//			(*Pierwsze szukanie*)
//			IF NOT bScrew1MinFound THEN															(*W1*)
//				IF ABS(ABS(lrStartPosition1FindingScrew)-ABS(Screwing1AxisRef.NcToPlc.ActPos))	>	100  THEN 
//					//IF lrScrewer1ActualTorque > (lrScrewer1MinTorqueWhenFindingScrew - 5) AND lrScrewer1ActualTorque < (lrScrewer1MaxTorqueWhenFindingScrew + 15) THEN		
////					IF diSensorHeightCV < -39000 THEN		(*W2*) //Dla Słoików 300ml
//					IF diSensorHeightCV < ((lrScrewerMaxSensorHeightWhenFindingScrew+lrScrewerMinSensorHeightWhenFindingScrew)/2) THEN		(*W2*) //Dla Słoików 300ml						
//						bScrew1MinFound						:=	TRUE;
//						lrStartPosition1FindingScrew 		:=	Screwing1AxisRef.NcToPlc.ActPos;
//					END_IF	
//				END_IF
//			END_IF
//			IF NOT bScrew2MinFound THEN															(*W1*)
//				IF ABS(ABS(lrStartPosition2FindingScrew)-ABS(Screwing2AxisRef.NcToPlc.ActPos))	>	100  THEN 
////					IF diSensorHeightCV < -39000 THEN		(*W2*)	//Dla Słoików 300ml	
//					IF diSensorHeightCV < ((lrScrewerMaxSensorHeightWhenFindingScrew+lrScrewerMinSensorHeightWhenFindingScrew)/2) THEN		(*W2*)	//Dla Słoików 300ml	
//						bScrew2MinFound						:=	TRUE;	
//						lrStartPosition2FindingScrew 		:=	Screwing2AxisRef.NcToPlc.ActPos;
//					END_IF	
//				END_IF	
//			END_IF
//			lrScrewerOffsetSensorHeightWhenFindingScrew	:=	((lrScrewerMaxSensorHeightWhenFindingScrew+lrScrewerMinSensorHeightWhenFindingScrew)/2)
//																+(lrScrewerMinSensorHeightWhenFindingScrew-lrScrewerMaxSensorHeightWhenFindingScrew)/6;
			
//			(*Drugie szukanie*)																					(*W3*)
//			IF bScrew1MinFound AND ABS(ABS(lrStartPosition1FindingScrew)-ABS(Screwing1AxisRef.NcToPlc.ActPos))	>	10  THEN 
				
//				IF diSensorHeightCV > lrScrewerOffsetSensorHeightWhenFindingScrew THEN		(*W4*)	//Dla Słoików 300ml
//					bScrew1Found						:=	TRUE;
//					mcScrewer1MoveRelative.Execute		:=	FALSE;
//					lrStartPosition1FindingScrew 		:=	Screwing1AxisRef.NcToPlc.ActPos;
//				END_IF
//			END_IF																								(*W3*)
//			IF bScrew2MinFound AND ABS(ABS(lrStartPosition2FindingScrew)-ABS(Screwing2AxisRef.NcToPlc.ActPos))	>	10  THEN 
//				IF diSensorHeightCV > ((lrScrewerMaxSensorHeightWhenFindingScrew+lrScrewerMinSensorHeightWhenFindingScrew)/2) THEN		(*W4*)	//Dla Słoików 300ml
//					bScrew2Found						:=	TRUE;
//					mcScrewer2MoveRelative.Execute		:=	FALSE;
//					lrStartPosition2FindingScrew 		:=	Screwing1AxisRef.NcToPlc.ActPos;
//				END_IF
//			END_IF

//			IF bScrew1Found  THEN

//				uiScrewing1TorqueControl		:=	6000;
//				mcScrewer1Stop.Execute			:=	TRUE;
				
//			END_IF
			
//			IF bScrew2Found  THEN

//				uiScrewing2TorqueControl		:=	6000;
//				mcScrewer2Stop.Execute			:=	TRUE;
//			END_IF			
			
//			IF	((bScrew1Found AND mcScrewer1Stop.Done) OR NOT bRun1 OR mcScrewer1MoveRelative.Done) AND
//				((bScrew2Found AND mcScrewer2Stop.Done) OR NOT bRun2 OR mcScrewer2MoveRelative.Done)
//			THEN
//				 mcScrewer1MoveRelative.Execute 	:=	FALSE;
//				 mcScrewer1Stop.Execute				:=	FALSE;
//				 mcScrewer2MoveRelative.Execute 	:=	FALSE;		
//				 mcScrewer2Stop.Execute				:=	FALSE;	 
//				 iFindingScrewCASE					:=	iFindingScrewCASE	+	10;	
//			END_IF
			
//		50: 
//			IF tonFindingScrewDelay.Q THEN
// 				iFindingScrewCASE					:=	iFindingScrewCASE	+	10;						
//			END_IF




END_IF
END_ACTION

ACTION Running6ScrewingMomentaryMode:
IF mcScrewer1TorqueControl.Error OR mcScrewer1MoveVelocity.Error OR mcScrewer1MoveVelocity2.Error
	 OR mcScrewer1MoveVelocity3.Error OR mcScrewer1MoveRelative.Error OR mcScrewer1MoveAbsolute.Error THEN
	bTest:= TRUE;
END_IF
tonInEndVelocity(IN:=mcScrewer1MoveContinuousRel.InEndVelocity, PT:=T#2MS);


				(********** TRYB MOMENTOWY **********)
					CASE iScrewingCase OF 	
					0:
						(* Wersja 2 - gearowanie Multi Master***************************************************************) 
						IF iTool <> 2 THEN
							bGripper1Actuator						:=	bRun1; // Ponowne załączanie chwytaków, dlatego
							bGripper2Actuator						:=	bRun2; // że jest możliwa duża ilość opcji
						ELSE
							bGripper1Actuator						:=	FALSE; // Ponowne załączanie chwytaków, dlatego
							bGripper2Actuator						:=	FALSE;
						END_IF
						//Właczenie sięcia osi
						mcHeightGearInMultiMaster.Enable			:=	TRUE;				
						//Jak osie spięte to początek kręcenia
						IF	mcHeightGearInMultiMaster.InGear AND 
							(tonGripper1Delay.Q OR sTool = 'ksztaltowa/do kulek' OR NOT bRun1) AND (tonGripper2Delay.Q OR sTool = 'ksztaltowa/do kulek'  OR NOT bRun2) // ton'y powinny być już wczesniej załączone jeżeli były chwytaki	
						THEN
							//Bloczek obrotu o zadany kąt i kontynuowania ruchu z zadaną prędkością
							mcScrewer1MoveContinuousRel.Execute				:= bRun1;
							//Kąt zmodyfikowany o różnicę między pozycją zatrzymania zakręcarki a pozycją wykrycia gwintu
							mcScrewer1MoveContinuousRel.Distance			:= Screwing1AxisRef.NcToPlc.ActPos - lrStartPosition1 + lrPackageTurnoversToFullScrewed*360.0-30.0;

							//DODAĆ ZABEZPIECZENIE JAK WYJDZIE ABSURDALNY KĄT
							
							//Prędkość na wyjściu z bloczka 120RPM - Inercja zakręcarki jest rozsądna
							mcScrewer1MoveContinuousRel.EndVelocity			:= 360*2;
							//Prędkość zakręcania wg parametrów
							mcScrewer1MoveContinuousRel.Velocity			:= (lrScrewerSpeed);
														
							iScrewingCase									:=	25;//iScrewingCase + 10;			
						END_IF
						
					10:	
					
						IF ABS(ABS(lrStartPosition1)-ABS(Screwing1AxisRef.NcToPlc.ActPos))>(lrPackageTurnoversToFullScrewed*360.0-90.0)  THEN 
							mcScrewer1MoveVelocity.Execute					:= FALSE;
							mcScrewer1MoveVelocity2.Execute					:= bRun1;
							mcScrewer1MoveVelocity2.Velocity				:= 360;
							uiScrewing1TorqueControl						:=	60000;
						//	mcScrewer1TorqueControl.Torque					:=	-5000;		
						//	mcScrewer1TorqueControl.TorqueRamp				:=	80000;	
							mcScrewer1TorqueControl.VelocityLimitHigh		:=	360;//(lrScrewerSpeed)/3.0;
							mcScrewer1TorqueControl.VelocityLimitLow		:=	-360;//-(lrScrewerSpeed)/3.0;
							iScrewingCase									:=	iScrewingCase + 10;	
						END_IF	
							
//						IF ABS(ABS(lrStartPosition2)-ABS(Screwing2AxisRef.NcToPlc.ActPos))>(lrPackageTurnoversToFullScrewed*360.0/7)  THEN 
//							mcScrewer2TorqueControl.Torque					:=	-9;		
//							mcScrewer2TorqueControl.TorqueRamp				:=	1500;					
//							mcScrewer2TorqueControl.VelocityLimitLow		:=	-4000;
//						END_IF	
					20:	
						mcScrewer1MoveVelocity2.Execute					:= FALSE;
						IF ABS(ABS(lrStartPosition1)-ABS(Screwing1AxisRef.NcToPlc.ActPos))>(lrPackageTurnoversToFullScrewed*360.0-15.0)  THEN
							mcScrewer1MoveVelocity2.Execute					:= FALSE;
							mcScrewer1TorqueControl.Execute					:=	bRun1;
							mcScrewer1TorqueControl.Torque					:=	(INT_TO_UINT(iScrewer1SetTorque)+iScrewer1AddTorque);		
						//	mcScrewer1TorqueControl.TorqueRamp				:=	4000;					
						//	mcScrewer1TorqueControl.VelocityLimitLow		:=	- 10;//(lrScrewerSpeed)/3.0;
							iScrewingCase									:=	iScrewingCase + 10;	
						END_IF	
							
						IF ABS(ABS(lrStartPosition2)-ABS(Screwing2AxisRef.NcToPlc.ActPos))>(lrPackageTurnoversToFullScrewed*360.0/6)  THEN 
							mcScrewer2TorqueControl.Torque					:=	(INT_TO_UINT(iScrewer2SetTorque)+iScrewer2AddTorque);		
							mcScrewer2TorqueControl.TorqueRamp				:=	4000;					
							mcScrewer2TorqueControl.VelocityLimitLow		:=	-(lrScrewerSpeed);
						END_IF	
						
					25:
						//Jak dojedzie do końca ruchu
						IF mcScrewer1MoveContinuousRel.InEndVelocity AND tonInEndVelocity.Q THEN
							mcScrewer1MoveContinuousRel.Execute				:= FALSE;
							//Przygotowanie trybu momentowego
							mcScrewer1TorqueControl.Execute					:=	bRun1;
							mcScrewer1TorqueControl.Torque					:=	(INT_TO_UINT(iScrewer1SetTorque)+iScrewer1AddTorque);	
							mcScrewer1TorqueControl.TorqueRamp				:=	8000;
							mcScrewer1TorqueControl.VelocityLimitHigh		:=	360*2;//(lrScrewerSpeed)/3.0;
							mcScrewer1TorqueControl.VelocityLimitLow		:=	-360*2;//-(lrScrewerSpeed)/3.0;	
							iScrewingCase									:=	30;//iScrewingCase + 10;	
						END_IF
	
					30:
						IF tonMomentaryScrewing1Timer.Q OR bWarning1 THEN
							mcScrewer1Stop.Execute				:=	TRUE;
							bGripper1Actuator					:=	FALSE;
							mcScrewer1TorqueControl.Execute		:=	FALSE;
							uiScrewing1TorqueControl			:=	0;
							bScrewed1							:=	TRUE;	
						END_IF
						IF tonMomentaryScrewing2Timer.Q OR bWarning2 THEN
							mcScrewer2Stop.Execute				:=	TRUE;
							bGripper2Actuator					:=	FALSE;
							mcScrewer2TorqueControl.Execute		:=	FALSE;
							uiScrewing2TorqueControl			:=	0;
							bScrewed2							:=	TRUE;		
						END_IF
				
						// Warunki zakręcenia zaleznie od uruchomionej zakręcarki
						IF (bScrewed1 OR NOT bRun1) AND (bScrewed2 OR NOT bRun2) AND
							(mcScrewer1Stop.Done OR NOT mcScrewer1Stop.Execute) AND 
							(mcScrewer2Stop.Done OR NOT mcScrewer2Stop.Execute) THEN
								mcScrewer1Stop.Execute			:= FALSE;
								mcScrewer2Stop.Execute			:= FALSE;
								iScrewingCase					:= iScrewingCase + 10;		
						END_IF
					40:
						(* Rozgearowanie osi *)
						mcHeightGearOut.Execute				:=	TRUE;
						mcHeightGearInMultiMaster.Enable	:=	FALSE;
	
						IF  mcHeightGearOut.Done THEN
							mcHeightGearOut.Execute					:= FALSE;
							eRunningState							:= E_GripperScrewer.eHolding;	
							iScrewingCase							:= 0;	
						END_IF			
					END_CASE
END_ACTION

ACTION Running6ScrewingPositionTorqueMode:
				(********* TRYB POZYCYJNY  *********)
				
				lrPackageThreadPitch;	
				(*Wymuszanie zwiększonego momentu przez 1/4 całego zakręcania*)
				IF ABS(ABS(lrStartPosition1)-ABS(Screwing1AxisRef.NcToPlc.ActPos))>(lrPackageTurnoversToFullScrewed*360.0/7)  THEN 
							uiScrewing1TorqueControl			:=	(INT_TO_UINT(iScrewer1SetTorque+3)*10)+(iScrewer1AddTorque*10);	
				ELSE		uiScrewing1TorqueControl			:=	6000;
				END_IF
				//uiScrewing1TorqueControl			:=	(INT_TO_UINT(iScrewerSetTorque+3)*10)+iScrewer1AddTorque;	
				(*Wymuszanie zwiększonego momentu przez 1/4 całego zakręcania*)
				IF ABS(ABS(lrStartPosition2)-ABS(Screwing2AxisRef.NcToPlc.ActPos))>(lrPackageTurnoversToFullScrewed*360.0/7)  THEN 
							uiScrewing2TorqueControl			:=	(INT_TO_UINT(iScrewer2SetTorque+3)*10)+(iScrewer2AddTorque*10);		
				ELSE		uiScrewing2TorqueControl			:=	6000;
				END_IF	

					CASE iScrewingCase OF 	
					0:
						(* Wersja 2 - gearowanie Multi Master***************************************************************) 
						IF iTool <> 2 THEN
							bGripper1Actuator						:=	bRun1; // Ponowne załączanie chwytaków, dlatego
							bGripper2Actuator						:=	bRun2; // że jest możliwa duża ilość opcji
						ELSE
							bGripper1Actuator						:=	FALSE; // Ponowne załączanie chwytaków, dlatego
							bGripper2Actuator						:=	FALSE; // że jest możliwa duża ilość opcji
						END_IF
						mcHeightGearInMultiMaster.Enable			:=	TRUE;				
						(* Start zakręcania *)
						IF	mcHeightGearInMultiMaster.InGear AND 
							(tonGripper1Delay.Q OR sTool = 'ksztaltowa/do kulek' OR NOT bRun1) AND (tonGripper2Delay.Q OR sTool = 'ksztaltowa/do kulek' OR NOT bRun2) // ton'y powinny być już wczesniej załączone jeżeli były chwytaki	
						THEN

							CASE iScrewing2Case OF 	
								
							0:
							
								mcScrewer1MoveVelocity2.Velocity		:=	5000;
								mcScrewer1MoveVelocity2.Execute		:=	bRun1;
								mcScrewer1MoveVelocity2.Direction	:=	MC_Positive_Direction;
																				
								mcScrewer2MoveVelocity2.Velocity		:=	5000;
								mcScrewer2MoveVelocity2.Execute		:=	bRun2;
								mcScrewer2MoveVelocity2.Direction	:=	MC_Positive_Direction;	
	
								iScrewing2Case						:=	iScrewing2Case + 10;										
							
							10:
								mcScrewer1MoveVelocity2.Execute		:=	FALSE;
								mcScrewer2MoveVelocity2.Execute		:=	FALSE;
							
								iScrewing2Case						:=	iScrewing2Case + 10;
	
							20:
							
								mcScrewer1MoveVelocity.Velocity		:=	lrScrewerSpeed;		
								mcScrewer1MoveVelocity.Direction	:=	MC_Positive_Direction;	
								IF ABS(ABS(lrStartPosition1)-ABS(Screwing1AxisRef.NcToPlc.ActPos))>(lrPackageTurnoversToFullScrewed*360.0/7)  THEN 									
									mcScrewer1MoveVelocity.Execute		:=	bRun1;									
								END_IF
								mcScrewer2MoveVelocity.Velocity		:=	lrScrewerSpeed;	
								mcScrewer1MoveVelocity.Direction		:=	MC_Positive_Direction;	
								IF ABS(ABS(lrStartPosition2)-ABS(Screwing2AxisRef.NcToPlc.ActPos))>(lrPackageTurnoversToFullScrewed*360.0/7)  THEN 
	
									mcScrewer2MoveVelocity.Execute		:=	bRun2;
								END_IF			

								IF (mcScrewer1MoveVelocity.Execute OR NOT bRun1) AND (mcScrewer2MoveVelocity.Execute OR NOT bRun2) THEN
									iScrewing2Case					:= 0	;
									iScrewingCase					:= iScrewingCase + 10;		
								END_IF
								
							END_CASE
							
						END_IF
						
					10:	
					
						(*Zmniejszanie prędkości jeżeli jest już przytrzymanie*)
						IF tonTightScrewing1Timer.ET > T#0S AND Screwing1AxisRef.NcToPlc.ActVelo < 10 THEN
							//mcScrewer1MoveVelocity.Execute		:= FALSE;
							//mcScrewer1MoveVelocity2.Execute		:= FALSE;
							
							//mcScrewer1MoveVelocity3.Velocity	:=	10;
							//mcScrewer1MoveVelocity3.Execute		:=	bRun1;
							//mcScrewer1MoveVelocity3.Direction	:=	MC_Positive_Direction;		

							rScrewing1ProportionalGain	:= 0;
							//rScrewing2ProportionalGain	:= 0;												
						END_IF
						
						IF tonTightScrewing2Timer.ET > T#0S AND Screwing2AxisRef.NcToPlc.ActVelo < 10 THEN
							//mcScrewer2MoveVelocity.Execute		:= FALSE;
							//mcScrewer2MoveVelocity2.Execute		:= FALSE;
							
							//mcScrewer2MoveVelocity3.Velocity	:=	10;
							//mcScrewer2MoveVelocity3.Execute		:=	bRun1;
							//mcScrewer2MoveVelocity3.Direction	:=	MC_Positive_Direction;		

							//rScrewing1ProportionalGain	:= 0;
							rScrewing2ProportionalGain	:= 0;												
						END_IF					
					
						(* Sprawdzanie czy osiągnięto moment lub zbyt długie zakracanie*)				
						IF tonTightScrewing1Timer.Q OR bWarning1 THEN
							bGripper1Actuator					:=	FALSE;
							bScrewed1							:=	TRUE;	
						END_IF
						IF tonTightScrewing2Timer.Q OR bWarning2 THEN
							bGripper2Actuator					:=	FALSE;
							bScrewed2							:=	TRUE;		
						END_IF
	
						IF tonTightScrewing1TimerAndOpenedGripper.Q THEN
							mcScrewer1Stop.Execute				:=	TRUE;
							mcScrewer1MoveVelocity.Execute		:=	FALSE;
							mcScrewer1MoveVelocity2.Execute		:=	FALSE;
							mcScrewer1MoveVelocity3.Execute		:=	FALSE;							
							uiScrewing1TorqueControl			:=	0;
						END_IF
						IF tonTightScrewing2TimerAndOpenedGripper.Q THEN
							mcScrewer2Stop.Execute				:=	TRUE;
							mcScrewer2MoveVelocity.Execute		:=	FALSE;
							mcScrewer2MoveVelocity2.Execute		:=	FALSE;	
							mcScrewer2MoveVelocity3.Execute		:=	FALSE;							
							uiScrewing2TorqueControl			:=	0;
						END_IF
					
						// Warunki zakręcenia zaleznie od uruchomionej zakręcarki
						IF (tonTightScrewing1TimerAndOpenedGripper.Q OR NOT bRun1) AND (tonTightScrewing2TimerAndOpenedGripper.Q OR NOT bRun2) AND
							(mcScrewer1Stop.Done OR NOT mcScrewer1Stop.Execute) AND 
							(mcScrewer2Stop.Done OR NOT mcScrewer2Stop.Execute) THEN
								mcScrewer1Stop.Execute			:= FALSE;
								mcScrewer2Stop.Execute			:= FALSE;
								iScrewingCase					:= iScrewingCase + 10;		
						END_IF
						
					20:
						(* Rozgearowanie osi *)
						mcHeightGearOut.Execute				:=	TRUE;
						mcHeightGearInMultiMaster.Enable	:=	FALSE;
	
						IF  mcHeightGearOut.Done THEN
							mcHeightGearOut.Execute					:= FALSE;
							eRunningState							:= E_GripperScrewer.eHolding;	
							iScrewingCase							:= 0;	
						END_IF			
					END_CASE
END_ACTION

ACTION Screwer1ControlBlocks:
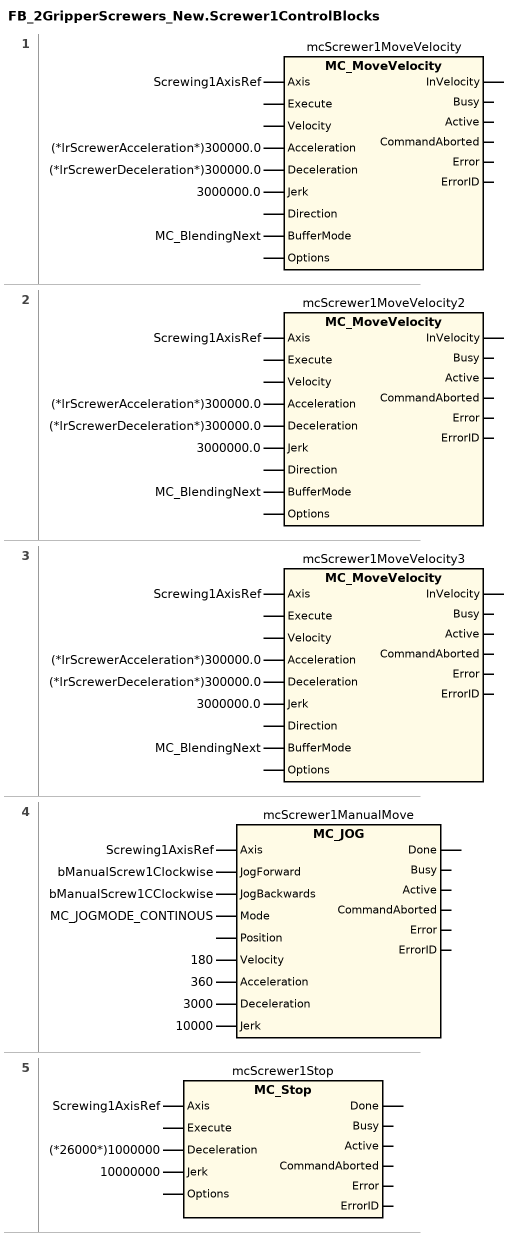
// NETWORK 1
mcScrewer1MoveVelocity(
    Axis := Screwing1AxisRef,
    Acceleration := (*lrScrewerAcceleration*)300000.0,
    Deceleration := (*lrScrewerDeceleration*)300000.0,
    Jerk := 3000000.0,
    BufferMode := MC_BlendingNext); // MC_MoveVelocity

// NETWORK 2
mcScrewer1MoveVelocity2(
    Axis := Screwing1AxisRef,
    Acceleration := (*lrScrewerAcceleration*)300000.0,
    Deceleration := (*lrScrewerDeceleration*)300000.0,
    Jerk := 3000000.0,
    BufferMode := MC_BlendingNext); // MC_MoveVelocity

// NETWORK 3
mcScrewer1MoveVelocity3(
    Axis := Screwing1AxisRef,
    Acceleration := (*lrScrewerAcceleration*)300000.0,
    Deceleration := (*lrScrewerDeceleration*)300000.0,
    Jerk := 3000000.0,
    BufferMode := MC_BlendingNext); // MC_MoveVelocity

// NETWORK 4
mcScrewer1ManualMove(
    Axis := Screwing1AxisRef,
    JogForward := bManualScrew1Clockwise,
    JogBackwards := bManualScrew1CClockwise,
    Mode := MC_JOGMODE_CONTINOUS,
    Velocity := 180,
    Acceleration := 360,
    Deceleration := 3000,
    Jerk := 10000); // MC_JOG

// NETWORK 5
mcScrewer1Stop(Axis := Screwing1AxisRef, Deceleration := (*26000*)1000000, Jerk := 10000000); // MC_Stop

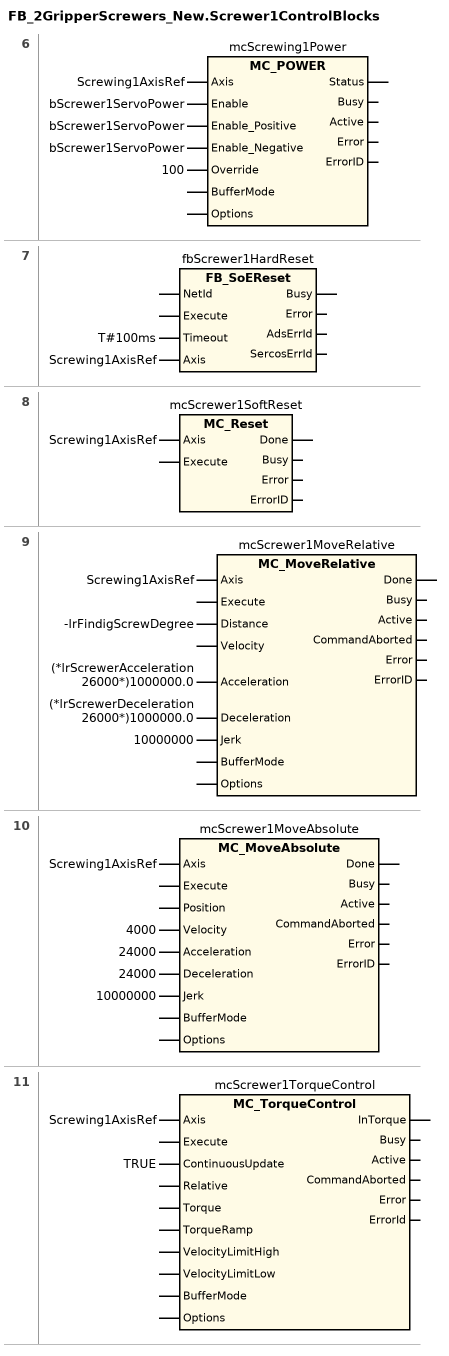
// NETWORK 6
mcScrewing1Power(
    Axis := Screwing1AxisRef,
    Enable := bScrewer1ServoPower,
    Enable_Positive := bScrewer1ServoPower,
    Enable_Negative := bScrewer1ServoPower,
    Override := 100); // MC_POWER

// NETWORK 7
fbScrewer1HardReset(Timeout := T#100ms, Axis := Screwing1AxisRef); // FB_SoEReset

// NETWORK 8
mcScrewer1SoftReset(Axis := Screwing1AxisRef); // MC_Reset

// NETWORK 9
mcScrewer1MoveRelative(
    Axis := Screwing1AxisRef,
    Distance := -lrFindigScrewDegree,
    Acceleration := (*lrScrewerAcceleration 26000*)1000000.0,
    Deceleration := (*lrScrewerDeceleration 26000*)1000000.0,
    Jerk := 10000000); // MC_MoveRelative

// NETWORK 10
mcScrewer1MoveAbsolute(
    Axis := Screwing1AxisRef,
    Velocity := 4000,
    Acceleration := 24000,
    Deceleration := 24000,
    Jerk := 10000000); // MC_MoveAbsolute

// NETWORK 11
mcScrewer1TorqueControl(Axis := Screwing1AxisRef, ContinuousUpdate := TRUE); // MC_TorqueControl

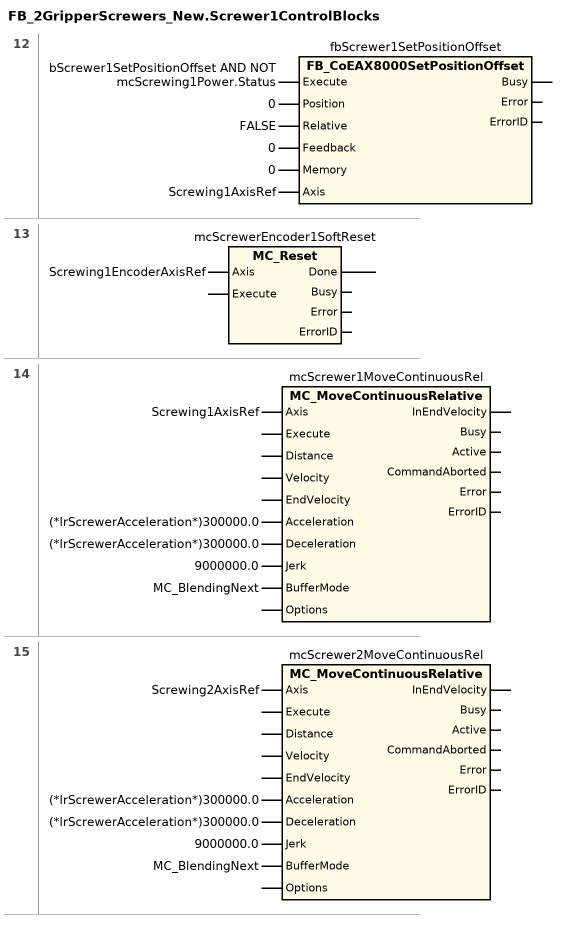
// NETWORK 12
fbScrewer1SetPositionOffset(
    Execute := bScrewer1SetPositionOffset AND NOT mcScrewing1Power.Status,
    Position := 0,
    Relative := FALSE,
    Feedback := 0,
    Memory := 0,
    Axis := Screwing1AxisRef); // FB_CoEAX8000SetPositionOffset

// NETWORK 13
mcScrewerEncoder1SoftReset(Axis := Screwing1EncoderAxisRef); // MC_Reset

// NETWORK 14
mcScrewer1MoveContinuousRel(
    Axis := Screwing1AxisRef,
    Acceleration := (*lrScrewerAcceleration*)300000.0,
    Deceleration := (*lrScrewerAcceleration*)300000.0,
    Jerk := 9000000.0,
    BufferMode := MC_BlendingNext); // MC_MoveContinuousRelative

// NETWORK 15
mcScrewer2MoveContinuousRel(
    Axis := Screwing2AxisRef,
    Acceleration := (*lrScrewerAcceleration*)300000.0,
    Deceleration := (*lrScrewerAcceleration*)300000.0,
    Jerk := 9000000.0,
    BufferMode := MC_BlendingNext); // MC_MoveContinuousRelative
END_ACTION

ACTION Screwer2ControlBlocks:
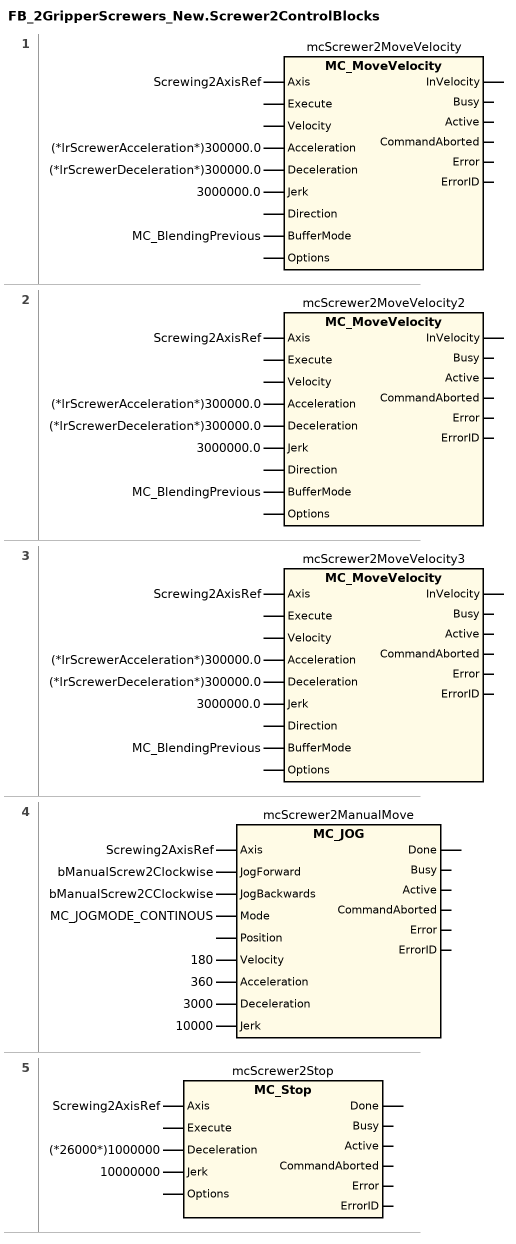
// NETWORK 1
mcScrewer2MoveVelocity(
    Axis := Screwing2AxisRef,
    Acceleration := (*lrScrewerAcceleration*)300000.0,
    Deceleration := (*lrScrewerDeceleration*)300000.0,
    Jerk := 3000000.0,
    BufferMode := MC_BlendingPrevious); // MC_MoveVelocity

// NETWORK 2
mcScrewer2MoveVelocity2(
    Axis := Screwing2AxisRef,
    Acceleration := (*lrScrewerAcceleration*)300000.0,
    Deceleration := (*lrScrewerDeceleration*)300000.0,
    Jerk := 3000000.0,
    BufferMode := MC_BlendingPrevious); // MC_MoveVelocity

// NETWORK 3
mcScrewer2MoveVelocity3(
    Axis := Screwing2AxisRef,
    Acceleration := (*lrScrewerAcceleration*)300000.0,
    Deceleration := (*lrScrewerDeceleration*)300000.0,
    Jerk := 3000000.0,
    BufferMode := MC_BlendingPrevious); // MC_MoveVelocity

// NETWORK 4
mcScrewer2ManualMove(
    Axis := Screwing2AxisRef,
    JogForward := bManualScrew2Clockwise,
    JogBackwards := bManualScrew2CClockwise,
    Mode := MC_JOGMODE_CONTINOUS,
    Velocity := 180,
    Acceleration := 360,
    Deceleration := 3000,
    Jerk := 10000); // MC_JOG

// NETWORK 5
mcScrewer2Stop(Axis := Screwing2AxisRef, Deceleration := (*26000*)1000000, Jerk := 10000000); // MC_Stop

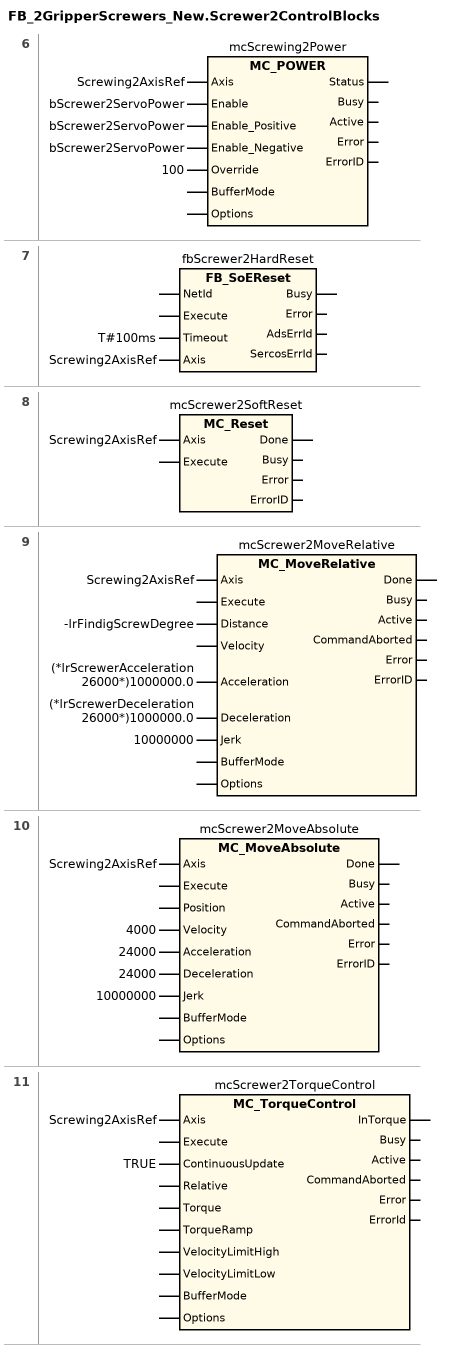
// NETWORK 6
mcScrewing2Power(
    Axis := Screwing2AxisRef,
    Enable := bScrewer2ServoPower,
    Enable_Positive := bScrewer2ServoPower,
    Enable_Negative := bScrewer2ServoPower,
    Override := 100); // MC_POWER

// NETWORK 7
fbScrewer2HardReset(Timeout := T#100ms, Axis := Screwing2AxisRef); // FB_SoEReset

// NETWORK 8
mcScrewer2SoftReset(Axis := Screwing2AxisRef); // MC_Reset

// NETWORK 9
mcScrewer2MoveRelative(
    Axis := Screwing2AxisRef,
    Distance := -lrFindigScrewDegree,
    Acceleration := (*lrScrewerAcceleration 26000*)1000000.0,
    Deceleration := (*lrScrewerDeceleration 26000*)1000000.0,
    Jerk := 10000000); // MC_MoveRelative

// NETWORK 10
mcScrewer2MoveAbsolute(
    Axis := Screwing2AxisRef,
    Velocity := 4000,
    Acceleration := 24000,
    Deceleration := 24000,
    Jerk := 10000000); // MC_MoveAbsolute

// NETWORK 11
mcScrewer2TorqueControl(Axis := Screwing2AxisRef, ContinuousUpdate := TRUE); // MC_TorqueControl

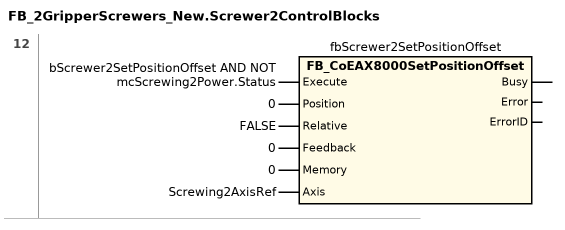
// NETWORK 12
fbScrewer2SetPositionOffset(
    Execute := bScrewer2SetPositionOffset AND NOT mcScrewing2Power.Status,
    Position := 0,
    Relative := FALSE,
    Feedback := 0,
    Memory := 0,
    Axis := Screwing2AxisRef); // FB_CoEAX8000SetPositionOffset
END_ACTION

ACTION Simulation:
(* Przyśpieszanie bloku gdy jest włączona symulacja*)

//tonSimulationScrewing1			(IN:=eRunningState=E_GripperScrewer.eScrewing 	AND bRun1 AND NOT bScrewed1 AND bSimulation,	PT:=T#0MS);
//tonSimulationScrewing2			(IN:=eRunningState=E_GripperScrewer.eScrewing 	AND bRun1 AND NOT bScrewed2 AND bSimulation,	PT:=T#0MS);

IF bSimulation THEN 			// Włączona symulacja
	tTooLongScrewing1 := T#250MS;
	tTooLongScrewing2 := T#250MS;	
ELSE							// Normalna praca
	tTooLongScrewing1 := T#2S; 	//Zmienić na 2
	tTooLongScrewing2 := T#2S;	//Zmienić na 2
END_IF
END_ACTION

ACTION Statistics:

IF LREAL_TO_INT(lrHeightEndScrewingPosition)<> LREAL_TO_INT(lrHeightReadyPosition) THEN
	rtrigCycleTimerRead(CLK:=LREAL_TO_INT(lrHeightActualPosition) = LREAL_TO_INT(lrHeightReadyPosition));
	IF rtrigCycleTimerRead.Q THEN
			tCycleTime:=tonCycleTimer.ET;
	END_IF
	tonCycleTimer(IN:=LREAL_TO_INT(lrHeightActualPosition) <> LREAL_TO_INT(lrHeightReadyPosition),PT:=T#1D);	
ELSE
	rtrigCycleTimerRead(CLK:=(eRunningState=E_GripperScrewer.eDone) OR (eRunningState=E_GripperScrewer.eNotDone));
	IF rtrigCycleTimerRead.Q THEN
		tCycleTime:=tonCycleTimer.ET;
	END_IF
	tonCycleTimer(IN:=eRunningState>E_GripperScrewer.eReady,PT:=T#1D);
END_IF
END_ACTION

ACTION Tools:
(*Narzędzia*)
AsToolDescription[0] := 'Głowica dwuszczękowa';
AsToolDescription[1] := 'Głowica trójszczękowa'; 
AsToolDescription[2] := 'Głowica kształtowa/do kulek';
AsToolDescription[3] := 'Głowica wbijająca'; 
AsToolDescription[4] := 'Głowica zasysająca';


(*Głowica wbijająca*)
IF iTool = 3 THEN
	bOptionCapPushingWithoutScrewing := TRUE;
ELSE
	bOptionCapPushingWithoutScrewing := FALSE;
END_IF

(*Przepisanie wybranego narzędzia do zmiennej typu string*)
(*!!!!! NIE ZMIENIAĆ OPISÓW, POWIĄZANE W PROGRAMIE !!!!!!*)
IF iTool = 0 THEN sTool := 'dwuszczekowa';			END_IF 
IF iTool = 1 THEN sTool := 'trojszczekowa';			END_IF
IF iTool = 2 THEN sTool := 'ksztaltowa/do kulek';	END_IF
IF iTool = 3 THEN sTool := 'wbijajaca';				END_IF
IF iTool = 4 THEN sTool := 'zasysajaca';			END_IF
END_ACTION

ACTION TorqueControl:

(*Konfiguracja MC_TorqueControl*)
//T_TorqueControlOptions;
mcScrewer1TorqueControl.Options.EnableManualTorqueStartValue := FALSE;//TRUE;
mcScrewer1TorqueControl.Options.ManualTorqueStartValue       := Screwing1AxisRef.NcToPlc.ActTorque;

mcScrewer2TorqueControl.Options.EnableManualTorqueStartValue := TRUE;
mcScrewer2TorqueControl.Options.ManualTorqueStartValue       :=  Screwing2AxisRef.NcToPlc.ActTorque;
END_ACTION

ACTION Warnings:
//Resetowanie warningów przy nastepnym cyklu

IF rtRun1.Q  OR rtRun2.Q THEN
	
	bWarning1			:=	FALSE;
	bWarning1A			:=	FALSE;
	bWarning1B			:=	FALSE;
	bWarning1C			:=	FALSE;
	bWarning1D			:=	FALSE;
	bWarning1E			:=	FALSE;	
	bWarning2			:=	FALSE;
	bWarning2A			:=	FALSE;
	bWarning2B			:=	FALSE;
	bWarning2C			:=	FALSE;
	bWarning2D			:=	FALSE;
	bWarning2E			:=	FALSE;
	udiWarningID		:=	0;
	sWarningDescription	:=	'';
END_IF
END_ACTION

END_FUNCTION_BLOCK

// ---- POUs/FB/FB_CatchStation.TcPOU
(*
Nazwa:			FB_CatchStation
Opis:			Chwytak pod stacjami 
Wersja:			v1.2
Data:			2025-07-08
Autor:			TW,DP
Urzadzenia:		Silownik chwytania, podnośnik JIESANG
Konfiguracja:	
Zmiany:
20250708 - Homing false po wyj. z Manual
20230222 - Zwieksozmny czas bledu 9

Info:
- dodano błędy od nastaw powyżej max i min (error 7 i 8)
- dodawno bHomingNeeded
- wylaczanie wyjść zmiana 2 wylaczanie wyjsc jak zniknie Enable
*)


FUNCTION_BLOCK FB_CatchStation
VAR_INPUT
	bEnable: BOOL;						//Zezwolenie na pracę
	bEStop:BOOL;						//Stop Awaryjny włączony
	bRun:BOOL;							//Rozkaz łapania 
	bHoming:BOOL;						//Zezwolenie na wykonanie bazowania i pozycjonowania podajnika
	bHeightSet:BOOL;					//Ustaw wysokość
	bChangeover:BOOL;					//Ustawianie na zadaną wysokość do wymiany elementów formatowych
	bChangeOver2:BOOL;
	bIgnoreError:BOOL;					//Ignorowania błędów cyklu pracy
	bReset:BOOL;						//Reset błędu, jeśli w stanie "eError"
	nGripperScrewerPosition   	:LREAL; // Aktualna pozycja serwa od podnoszenia
	nSafetyScrewerPosition		:LREAL;	// zadana bezpieczna pozycja 
	bScrewerbError				:BOOL;  // Sygnał błędu od zakręcarki
	nPositionHeightSV:LREAL;			//Wysokość zadana na której ma znajdować się stacja
	bOpenedActuatorSensor:BOOL;			//Czujnik otwarcia siłownika łapania
	bClosedActuatorSensor:BOOL;			//Czujnik otwarcia siłownika łapania
	lrMaxHeight:LREAL;					//Maksymalna wysokość podnośnika chwytaka
	lrMinHeight:LREAL;					//Minimalna wysokość podnośnika chwytaka
	bManualMovement:BOOL;				//Zezwolenie na ruchy ręcznę
	bUnlockColision:BOOL:=FALSE;		//Odblokowywanie możliwośći kolizji
	bAlarmSVCVDiffHeightDisable:BOOL;	//Wyłączenie alarmu od rożnicy wysokości zadanej od aktualnej
	bNoLifter:BOOL;						//Podnośnik
	
	_HEIGHTMOTOR_ :BOOL;	
				
	rHeightMotorPositionOffset :REAL;		//Wysokość bazowani podnośnika
	udiHeightMotorEncoderCV		: UDINT;
	bHeightEncoderSetCDone		: BOOL;	

	_ALARMINFO_ :BOOL;
	iStationIndex:UDINT;					//Numer stacji 
	sStationName:WSTRING;					//Nazwa stacji	

	
END_VAR
VAR_OUTPUT
	eState: E_Station;						//Stan ogólny bloku
	eRunningState: E_CatchStationState;		//Stan wewnętrzny
	bError: BOOL;							//Błąd stacji
	nErrorNr: UDINT;						//Nr błędu podajnika platynek
	sErrorDescription:STRING(200);				//Opis błędu
	sErrorDescription2: STRING(200);				//Opis błędu 2
	sErrorStationName:STRING;				//Nazwa stacji
	udiStationID: UDINT;				// Nr stacji

	bCatchActuator:BOOL;					//Sterownie siłownika łapania opakowania
	bHeightMotorUp:BOOL;					//Sterowanie silnikiem podnośnika  - RUCH W GÓRĘ
	bHeightMotorDown:BOOL;					//Sterowanie silnikiem podnośnika  - RUCH W DÓŁ
	lrHeightMotorCV:LREAL;					//Aktualna pozycja podnośnika
	tCycleTime:TIME;
	bHomingDone:BOOL;						//Wymagane ponowne bazowanie (blad podczas bazowania lub stop awaryjny)
	bCycleDone:BOOL;
	bCycleNotDone:BOOL;
	
				
	udiHeightMotorEncoderSetCV	: UDINT;	
	bHeightEncoderSetC			: BOOL;		

END_VAR
VAR
	tonHeightNoChange: TON; 			//Timer wykrycia braku ruchu siłownika zmiany wysokości stacji
	nLastPositionHeightCV: LREAL;		//Pozycja podnośnika w poprzednim cyklu programu
	tonErrorHeightChange: TON; 			//Timer błędu podnośnika
	// Czas zadziałania siłownika
	tonCatchingTime: TON;
	// Timer blokady otwierania chwytaka
	tonOpeningBlocked: TON;
	rtEncoderHomed:R_TRIG;
	tonCycleTimer:TON;
	rtrigCycleTimerRead:R_TRIG;
	
	tofMotorUpPermition: TOF;
	tofMotorDownPermition: TOF;
	tonLimitPosMinReachedDelay: TON;
	tonLimitPosMaxReachedDelay: TON;
	tonMaxHeight		: TON;
	tonMinHeight		: TON;
	tonSVCVDiffHeight	: TON;
	
	//Podnośnik Jiesang	
	fbHeightMotorEncoder: FB_JiesangActuatorEncoderModul;	// Blok enkodera podnośnika chwytaka stabilizującego pod zakręcarką	
	bHeightMotorEncoderCounterReset:BOOL; 				//Sygnał resetu enkodera
	bHeightMotorEncoderHomed:BOOL;						//Informacja od enkodera że jest zbazowany

	eLastState: E_Station;							//Stan ogólny bloku
	eLastRunningState: E_CatchStationState;			//Stan podbloku
	eLastStateTemp: E_Station;						//Stan ogólny bloku
	eLastRunningStateTemp: E_CatchStationState;		//Stan podbloku
	bStateError: BOOL;

	tonStopping: TON;
	tofHeightMotorDown: TOF;
	iCaseChangeover: INT;
	tonChangeOverLimitPosMinReachedDelay: TON;
	tonChangeoverLimitPosMaxReachedDelay: TON;
	
	//Zmienne od EVENTLOGGER
	bAlarmInit 						: BOOL := TRUE; 
	nAlarmNumerator					: INT;
	arfbAlarm						: ARRAY[0..19] OF  FB_TcAlarm;		//Tablica bloczków błędów
	fbSourceInfo 					: FB_TcSourceInfo;
	iSourceInfo						: I_TcSourceInfo;
	sAlarmTest						: STRING;
	//Koniec zmiennych od EVENTLOGGER
END_VAR

VAR_IN_OUT
	bManualCatchActuator:BOOL;		//Ruch ręczny siłownikiem podajnika platynek
	bManualHeightMotorUp:BOOL;			//Ruch ręczny podnośnika stacji w górę
	bManualHeightMotorDown:BOOL;		//Ruch ręczny podnośnika stacji w dół
END_VAR

HeightMotor();
ErrorHandling();
Control();
Changeover();
Statistics();
aStationID();
(*Zapisywanie ostatniego stanu*)
IF eLastStateTemp<>eState THEN
	eLastState := eLastStateTemp;
END_IF
eLastStateTemp := eState;
IF eLastRunningStateTemp<>eRunningState THEN
	eLastRunningState := eLastRunningStateTemp;
END_IF
eLastRunningStateTemp := eRunningState;
(*Koniec Zapisywanie ostatniego stanu*)


nLastPositionHeightCV:=lrHeightMotorCV;

ACTION aStationID:
udiStationID	:=	iStationIndex;
END_ACTION

ACTION Changeover:
tonChangeOverLimitPosMinReachedDelay(IN:=(lrHeightMotorCV<=lrMinHeight) AND bChangeover,PT:=T#2S);
tonChangeoverLimitPosMaxReachedDelay(IN:=(lrHeightMotorCV>=lrMaxHeight) AND bChangeover,PT:=T#2S);


//Przeniesione do PreparingToDisabled
(*CASE iCaseChangeover OF
	
	0: //Włączenie ustawiania
		IF bChangeover THEN
			iCaseChangeover := iCaseChangeover + 10;
			bHeightMotorDown:=FALSE;
			bHeightMotorUp:=FALSE;
		END_IF
		
	10: //Ustawianie stacji na wysokość 
		IF bHeightMotorEncoderHomed THEN
			bHeightMotorEncoderCounterReset	:=	FALSE;
			bHeightMotorUp					:=	lrHeightMotorCV	<=	200;
			bHeightMotorDown				:=	lrHeightMotorCV	>=	200;
			//Kiedy stacja osiągnie wysokość zadaną
			IF ABS(lrHeightMotorCV-nPositionHeightSV)<2 OR tonChangeoverLimitPosMaxReachedDelay.Q OR tonChangeOverLimitPosMinReachedDelay.Q  THEN
				bHeightMotorDown			:=	FALSE;
				bHeightMotorUp				:=	FALSE;
				iCaseChangeover 			:=	iCaseChangeover + 10;
			END_IF			
		ELSE
			bHeightMotorDown		:=	FALSE;
			bHeightMotorUp			:=	FALSE;
			iCaseChangeover 		:=  0;
		END_IF	
		
	20: //Czekanie na wyłączenie przezbrajania i ustawienie na odpowiednią wysokość z receptury
			IF NOT bChangeover THEN
				iCaseChangeover := iCaseChangeover + 10;
			END_IF
	30: //Ustawianie stacji na wysokość z receptury
		IF bHeightMotorEncoderHomed THEN
			bHeightMotorEncoderCounterReset	:=	FALSE;
			bHeightMotorUp					:=	lrHeightMotorCV	<=	nPositionHeightSV;
			bHeightMotorDown				:=	lrHeightMotorCV	>=	nPositionHeightSV;
			//Kiedy stacja osiągnie wysokość zadaną
			IF ABS(lrHeightMotorCV-nPositionHeightSV)<2 OR tonChangeoverLimitPosMaxReachedDelay.Q OR tonChangeOverLimitPosMinReachedDelay.Q  THEN
				bHeightMotorDown			:=	FALSE;
				bHeightMotorUp				:=	FALSE;
				iCaseChangeover 			:=	iCaseChangeover + 10;
			END_IF			
		ELSE
			bHeightMotorDown		:=	FALSE;
			bHeightMotorUp			:=	FALSE;
			iCaseChangeover 		:=  0;
		END_IF
	40: //Ustawianie stacji na wysokość z receptury	
		iCaseChangeover 		:=  0;

END_CASE
*)
END_ACTION

ACTION Control:

	(** TIMERY**)
	rtEncoderHomed(CLK:=bHeightMotorEncoderHomed,Q=>);
	tonHeightNoChange(IN:=((bHeightMotorUp OR bHeightMotorDown) AND (nLastPositionHeightCV=lrHeightMotorCV)), PT:=T#1S); 
	tonLimitPosMinReachedDelay(IN:=(lrHeightMotorCV<=lrMinHeight) AND eState=E_Station.eHoming,PT:=T#2S);
	tonLimitPosMaxReachedDelay(IN:=(lrHeightMotorCV>=lrMaxHeight) AND eState=E_Station.eHoming,PT:=T#2S);
	tonStopping(IN:=eState=E_Station.eStopping,PT:=T#2S);
	tofMotorUpPermition(IN:=bHeightMotorDown,PT:=T#250MS);
	tofMotorDownPermition(IN:=bHeightMotorUp ,PT:=T#250MS);	
	(*****Wyłączenie enable*****)
	IF NOT bEnable OR bChangeover THEN //Lub przezbrajania
		IF eState <> E_Station.eDisabled AND eState <> E_Station.ePreparingToDisable AND nGripperScrewerPosition>nSafetyScrewerPosition AND NOT bScrewerbError THEN
				eState 				:= E_Station.ePreparingToDisable; 
		END_IF	
	END_IF

	(*****Estop*****)
	IF NOT bEstop  THEN	
		IF eState <> E_Station.eAborted AND eState <> E_Station.eAborting AND eState <> E_Station.eDisabled THEN
				eState 				:= E_Station.eAborting; 
		END_IF
	END_IF

	CASE eState OF
	/////////////////////////////	
		E_Station.eDisabled: 					// Stan nieaktywnosci (Stacja wyłączona) 

			IF bEnable THEN
				eState 				:= E_Station.ePreparingToReady; 
			END_IF 
			
    /////////////////////////////	    
		E_Station.eAborted: 					// Stan bezpiecznego zatrzymania (po Abortingu) 

			IF bEStop THEN
				eState 				:= E_Station.ePreparingToReady;
			END_IF
			
	/////////////////////////////	
		E_Station.eAborting:                 	// Stan bezpiecznego zatrzymywania (po EStopie)

			bHeightMotorUp				:=	FALSE;
			bHeightMotorDown			:=	FALSE;
			eState := E_Station.eAborted;  
			eRunningState:=E_CatchStationState.eDisabled;
			
	/////////////////////////////			
		E_Station.eError:                 	 	// Stan błędu 	

			iCaseChangeover 		:=	0;
			IF bReset THEN
				eState 				:=	E_Station.eResetting;
			END_IF
						
	/////////////////////////////
		E_Station.eResetting:					// Stan resetowania bledu (po Errorze)
	
			bError := FALSE;

			IF NOT bError THEN
				nErrorNr 			:=	0;
   				sErrorDescription 	:=	'';
				eState 				:=	E_Station.ePreparingToReady;
			ELSE
				eState 				:=	E_Station.eError;
			END_IF
        
	/////////////////////////////
		E_Station.eManualMovement:     			// Stan ruchów manualnych  

			ManualMovements();
			//Wyjście z trybu serwisowego
			IF NOT bManualMovement THEN
				IF bHomingDone AND ABS(lrHeightMotorCV - nPositionHeightSV)> 2 THEN
					bHomingDone := FALSE;
				END_IF
				bCatchActuator				:=	FALSE;
				bHeightMotorUp				:=	FALSE;
				bHeightMotorDown			:=	FALSE;
				bManualCatchActuator		:=	bCatchActuator;
				eState:=E_Station.eReady;
			END_IF

	/////////////////////////////
		E_Station.eHoming:						// Stan bazowania 
	IF (nGripperScrewerPosition>nSafetyScrewerPosition AND NOT bScrewerbError) OR bManualMovement THEN  // co to za bzdura
			Homing();
			IF NOT bHoming AND NOT bHeightSet THEN // co to za bzdura
			   eState:=E_Station.ePreparingToReady;
			   	bHeightMotorDown:=FALSE;
				bHeightMotorUp:=FALSE;
			END_IF		
	END_IF		
	/////////////////////////////
		E_Station.eHomingDone:                  // Stan wykonania bazowania 
	
			bHeightMotorDown					:=	FALSE;
			bHeightMotorUp						:=	FALSE;
			bHeightMotorEncoderCounterReset		:=	FALSE;
			bHomingDone							:=	TRUE;
			IF NOT bHoming AND NOT bHeightSet THEN
			   eState:=E_Station.eReady;
			END_IF
			
	/////////////////////////////
		E_Station.ePreparingToReady:            // Stan przygotowywania do gotowosci (zawsze przed Ready)  
	
			bCatchActuator	:=	FALSE;
			eRunningState	:=	E_CatchStationState.eReady;
			eState			:=	E_Station.eReady;	
			
	/////////////////////////////
		E_Station.ePreparingToDisable:          // Stan przygotowywania do nieaktywnosci (po wyłączeniu Enable) 
  
			bCatchActuator:=FALSE;
			IF NOT bChangeOver THEN //Normalne wyłączenie
				bHeightMotorUp:=TRUE;
				bHeightMotorDown:=FALSE;	
				IF tonHeightNoChange.Q THEN
					bHeightMotorUp:=FALSE;
					eState:=E_Station.eDisabled;
					eRunningState:=E_CatchStationState.eDisabled;
				END_IF	
			ELSE //Wyłączenie z przebrajaniem na pozycje 200
				IF bHeightMotorEncoderHomed THEN
					bHeightMotorEncoderCounterReset	:=	FALSE;
					bHeightMotorUp					:=	lrHeightMotorCV	<=	150 AND NOT tofMotorUpPermition.Q;
					bHeightMotorDown				:=	lrHeightMotorCV	>=	150 AND NOT tofMotorDownPermition.Q;
					//Kiedy stacja osiągnie wysokość zadaną
					IF ABS(lrHeightMotorCV-150)<2 OR tonChangeoverLimitPosMaxReachedDelay.Q OR tonChangeOverLimitPosMinReachedDelay.Q  THEN
						bHeightMotorDown			:=	FALSE;
						bHeightMotorUp				:=	FALSE;
						eState						:=	E_Station.eDisabled;
						eRunningState				:=	E_CatchStationState.eDisabled;
					END_IF			
				ELSE
					bHeightMotorDown				:=	FALSE;
					bHeightMotorUp					:=	FALSE;
					eState								:=E_Station.eDisabled;
					eRunningState					:=	E_CatchStationState.eDisabled;
				END_IF	
			END_IF
				
	/////////////////////////////
		E_Station.eReady:						// Stan gotowosci 

			IF bRun AND NOT bCycleDone AND NOT bCycleNotDone THEN
				eState 				:= E_Station.eStarting; 
			END_IF
			IF bHoming OR bHeightSet OR bChangeover THEN
				eState 				:= E_Station.eHoming; 
			END_IF
			IF bManualMovement THEN
				//Jeśli przejście w tryb ruchów manualnych przepisz wszystkie stany siłowników sterowanych przez moduł
				//aby zapobiec ewentualnym kolizjom po wejściu w tryb serwisowy
				bManualCatchActuator		:= bCatchActuator;
				bManualHeightMotorUp		:= bHeightMotorUp;
				bManualHeightMotorDown		:= bHeightMotorDown;
				
				eState 						:= E_Station.eManualMovement; 
				eRunningState 				:= E_CatchStationState.eReady;
 
			END_IF
			IF NOT bRun THEN
				bCycleDone 			:= FALSE;
				bCycleNotDone 		:= FALSE;			
			END_IF
			
	/////////////////////////////
		E_Station.eStopping:					// Stan zatrzymywania 
					
			Running();
			IF bOpenedActuatorSensor OR tonStopping.Q THEN //NEW
				eState						:=	E_Station.eReady;
				eRunningState 				:=	E_CatchStationState.eReady;
			END_IF
			
	/////////////////////////////
		E_Station.eStarting:                  	// Stan uruchamiania (po Ready)
				
			eState					 := E_Station.eRunning; 

	/////////////////////////////
		E_Station.eRunning:               		// Stan wykonywania cyklu (po Startingu), w tym stanie osobny

			Running();
			IF NOT bRun THEN 					(*Przerywanie cyklu*)
				eState				:= E_Station.eStopping;
				bCycleNotDone		:= TRUE;
			END_IF
			(*IF bCycleDone OR bCycleNotDone THEN (*Cykl zakończony*)
				eState 				 := E_Station.eReady;
			END_IF*)						
		ELSE
		
		
	/////////////////////////////		
	END_CASE
END_ACTION

ACTION ErrorHandling:
// Alarm_0440	440	Error	Blokada otwarcia chwytaka - sprawdź czujnik
// Alarm_0441	441	Error	Blokada podnośnika lub brak zasilania - sprawdź czujnik lub odblokuj mechanicznie
// Alarm_0442	442	Error	Wartość zadana wysokości jest większa od maksymalnej - zmień ustawienia w recepturze {0}
// Alarm_0443	443	Error	Wartość zadana wysokości jest mniejsza od minimalnej - zmień ustawienia w recepturze {0}
// Alarm_0444	444	Error	Wartość aktualna jest zbyt różna od zadanej - zmień ustawienia w recepturze lub ustaw stację

IF bAlarmInit THEN
    bAlarmInit := FALSE; 
	fbSourceInfo.Clear();
	fbSourceInfo.sName:=wsLiteral_TO_UTF8(sStationName);//'Machine';
	fbSourceInfo.nId:=iStationIndex;//2700;
	// Alarm_0440	440	Error	Blokada otwarcia chwytaka - sprawdź czujnik
    arfbAlarm[0].CreateEx(stEventEntry := TC_EVENTS.AlarmClass.Alarm_0440, bWithConfirmation:= FALSE,  ipSourceInfo:= fbSourceInfo); 
	// Alarm_0441	441	Error	Blokada podnośnika lub brak zasilania - sprawdź czujnik lub odblokuj mechanicznie
	arfbAlarm[1].CreateEx(stEventEntry := TC_EVENTS.AlarmClass.Alarm_0441, bWithConfirmation:= FALSE,  ipSourceInfo:= fbSourceInfo);
	// Alarm_0442	442	Error	Wartość zadana wysokości jest większa od maksymalnej - zmień ustawienia w recepturze {0}
	arfbAlarm[2].CreateEx(stEventEntry := TC_EVENTS.AlarmClass.Alarm_0442, bWithConfirmation:= FALSE,  ipSourceInfo:= fbSourceInfo);
	// Alarm_0443	443	Error	Wartość zadana wysokości jest mniejsza od minimalnej - zmień ustawienia w recepturze {0}
	arfbAlarm[3].CreateEx(stEventEntry := TC_EVENTS.AlarmClass.Alarm_0443, bWithConfirmation:= FALSE,  ipSourceInfo:= fbSourceInfo);
	// Alarm_0444	444	Error	Wartość aktualna jest zbyt różna od zadanej - zmień ustawienia w recepturze lub ustaw stację
	arfbAlarm[4].CreateEx(stEventEntry := TC_EVENTS.AlarmClass.Alarm_0444, bWithConfirmation:= FALSE,  ipSourceInfo:= fbSourceInfo);
END_IF

//OBSŁUGA BŁĘDÓW PODAJNIKA PLATYNEK

//************LISTA BŁĘDÓW***************
bStateError:= (eState=E_Station.eError) OR (eState=E_Station.eResetting) OR bIgnoreError;




IF bEnable THEN
	// Alarm_0440	440	Error	Blokada otwarcia chwytaka - sprawdź czujnik
	//Error 1 - Blokada otwarcia chwytaka
	tonOpeningBlocked(IN:=NOT bCatchActuator AND NOT bOpenedActuatorSensor, PT:=T#3S);
	
	IF tonOpeningBlocked.Q THEN
		IF NOT arfbAlarm[0].bActive THEN
			arfbAlarm[0].Raise(nTimeStamp:=0);
		END_IF
	ELSE	
		IF  arfbAlarm[0].bActive AND bReset THEN
			arfbAlarm[0].Clear(nTimeStamp:=0, bResetConfirmation:= FALSE);
		END_IF
// 		sErrorDescription:='Blokada otwarcia chwytaka - sprawdź czujnik';
// 		bHeightMotorUp:=FALSE;
// 		bError := TRUE;
// 		nErrorNr:=281;	
// 		//nErrorNr := nErrorNr+iStationIndex;
	END_IF
	// Alarm_0441	441	Error	Blokada podnośnika lub brak zasilania - sprawdź czujnik lub odblokuj mechanicznie
	//Error 2 - podnośnik nie porusza się pomimo wysterowania 
	tonErrorHeightChange(IN:=(bHeightMotorUp OR bHeightMotorDown) AND nLastPositionHeightCV=lrHeightMotorCV AND NOT bNoLifter, PT:=T#3S);
	
	IF tonErrorHeightChange.Q THEN
		IF NOT arfbAlarm[1].bActive THEN
			bHeightMotorUp:=FALSE;
			bHeightMotorDown:=FALSE;
			arfbAlarm[1].Raise(nTimeStamp:=0);
		END_IF
	ELSE	
		IF  arfbAlarm[1].bActive AND bReset THEN
			arfbAlarm[1].Clear(nTimeStamp:=0, bResetConfirmation:= FALSE);
		END_IF
// 		bHeightMotorUp:=FALSE;
// 		bHeightMotorDown:=FALSE;
// 		bError := TRUE;
// 		nErrorNr:=282;
// 		//nErrorNr := nErrorNr+iStationIndex;
// 		sErrorDescription:='Blokada podnośnika lub brak zasilania - sprawdź czujnik lub odblokuj mechanicznie';	
	END_IF
	
	// Alarm_0442	442	Error	Wartość zadana wysokości jest większa od maksymalnej - zmień ustawienia w recepturze {0}
	//Error 3 - Bład nastaw max
	tonMaxHeight(IN:=nPositionHeightSV>lrMaxHeight+1 AND bHomingDone AND lrMaxHeight>0 AND eState=E_Station.eReady,PT:=T#30S);
	IF tonMaxHeight.Q THEN
		arfbAlarm[2].ipArguments.Clear() .AddLReal(lrMaxHeight);
		IF NOT arfbAlarm[2].bActive THEN
			bHeightMotorUp:=FALSE;
			bHeightMotorDown:=FALSE;
			arfbAlarm[2].Raise(nTimeStamp:=0);
		END_IF
	ELSE	
		IF  arfbAlarm[2].bActive AND bReset THEN
			arfbAlarm[2].Clear(nTimeStamp:=0, bResetConfirmation:= FALSE);
		END_IF	
// 		bHeightMotorUp:=FALSE;
// 		bHeightMotorDown:=FALSE;
// 		bError := TRUE;
// 		nErrorNr:=283;
// 		//nErrorNr := nErrorNr+iStationIndex;
// 		sErrorDescription:='Wartość zadana wysokości jest większa od maksymalnej - zmień ustawienia w recepturze';
// 		sErrorDescription2:=REAL_TO_STRING(LREAL_TO_INT(lrMaxHeight));
	END_IF
	// Alarm_0443	443	Error	Wartość zadana wysokości jest mniejsza od minimalnej - zmień ustawienia w recepturze {0}
	//Error 4 - Bład nastaw min
	tonMinHeight(IN:=nPositionHeightSV<lrMinHeight-1 AND bHomingDone AND lrMinHeight>0 AND eState=E_Station.eReady,PT:=T#30S);
	IF tonMinHeight.Q THEN
		arfbAlarm[3].ipArguments.Clear() .AddLReal(lrMinHeight);
		IF NOT arfbAlarm[3].bActive THEN
			bHeightMotorUp:=FALSE;
			bHeightMotorDown:=FALSE;
			arfbAlarm[3].Raise(nTimeStamp:=0);
		END_IF
	ELSE	
		IF  arfbAlarm[3].bActive AND bReset THEN
			arfbAlarm[3].Clear(nTimeStamp:=0, bResetConfirmation:= FALSE);
		END_IF
// 		bHeightMotorUp:=FALSE;
// 		bHeightMotorDown:=FALSE;
// 		bError := TRUE;
// 		nErrorNr:=284;
// 		//nErrorNr := nErrorNr+iStationIndex;
// 		sErrorDescription:='Wartość zadana wysokości jest mniejsza od minimalnej - zmień ustawienia w recepturze ';
// 		sErrorDescription2:=REAL_TO_STRING(LREAL_TO_INT(lrMinHeight));
	END_IF
	// Alarm_0444	444	Error	Wartość aktualna jest zbyt różna od zadanej - zmień ustawienia w recepturze lub ustaw stację
	//Error 5 - Bład zbyt dużej różnicy nastaw
	//tonSVCVDiffHeight(IN:=ABS(nPositionHeightSV-lrHeightMotorCV)>10 AND bHomingDone AND NOT bAlarmSVCVDiffHeightDisable AND eState=E_Station.eReady AND NOT bChangeOver2,PT:=T#5M);
	IF tonSVCVDiffHeight.Q THEN
		arfbAlarm[4].ipArguments.Clear() .AddLReal(nPositionHeightSV);
		IF NOT arfbAlarm[4].bActive THEN
			bHeightMotorUp:=FALSE;
			bHeightMotorDown:=FALSE;
			arfbAlarm[4].Raise(nTimeStamp:=0);
		END_IF
	ELSE	
		IF  arfbAlarm[4].bActive AND bReset THEN
			arfbAlarm[4].Clear(nTimeStamp:=0, bResetConfirmation:= FALSE);
		END_IF
// 		bHeightMotorUp:=FALSE;
// 		bHeightMotorDown:=FALSE;
// 		bError := TRUE;
// 		nErrorNr:=285;
// 		//nErrorNr := nErrorNr+iStationIndex;
// 		sErrorDescription:='Wartość aktualna jest zbyt różna od zadanej - zmień ustawienia w recepturze lub ustaw stację';
// 		sErrorDescription2:=REAL_TO_STRING(LREAL_TO_INT(nPositionHeightSV));
		
	END_IF	
		
	
	
ELSE
	bError := FALSE;
END_IF

	
//******************PRZEJŚCIE DO eERROR*****************************

IF bError AND NOT bStateError THEN
	IF eLastState = eRunning THEN
		bCycleNotDone := TRUE;
	END_IF
	eState := E_Station.eError;
END_IF

//****************WYŚWIETLANIE STATUSU BLEDU***********************

(*Wyświetlanie błedu na wyjściu*)
bError							:= FALSE;
FOR nAlarmNumerator := 0 TO 19 DO
	bError						:= bError OR arfbAlarm[nAlarmNumerator].bActive;
END_FOR

(*Przepisywanie nazwy stacji*)
sErrorStationName := WSTRING_TO_STRING(sStationName);


//Jezeli nie zbazowane to potrzebne bazowanie
IF NOT bHeightMotorEncoderHomed AND NOT bNoLifter  THEN
	bHomingDone:=FALSE;
END_IF
END_ACTION

ACTION HeightMotor:
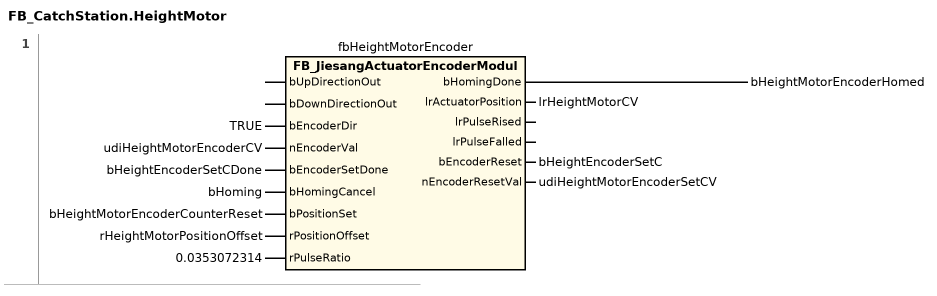
// NETWORK 1
fbHeightMotorEncoder(
    bEncoderDir := TRUE,
    nEncoderVal := udiHeightMotorEncoderCV,
    bEncoderSetDone := bHeightEncoderSetCDone,
    bHomingCancel := bHoming,
    bPositionSet := bHeightMotorEncoderCounterReset,
    rPositionOffset := rHeightMotorPositionOffset,
    rPulseRatio := 0.0353072314,
    lrActuatorPosition => lrHeightMotorCV,
    bEncoderReset => bHeightEncoderSetC,
    nEncoderResetVal => udiHeightMotorEncoderSetCV); // FB_JiesangActuatorEncoderModul
bHeightMotorEncoderHomed := fbHeightMotorEncoder.bHomingDone;
END_ACTION

ACTION Homing:
//BAZOWANIE
bCatchActuator:=FALSE;
	
//Uwaga nie zmieniać czasu bo jednocześnie dwie stację jadą do góry
tofHeightMotorDown(IN:=bHeightMotorDown, PT:=T#1S); //Zabezpieczenie przed zbyt szybkim przełączeniem pomiędzy Down a Up, bezpiecznieki sie palą, 


//Podnoszenie stacji do maksymalnej pozycji
IF NOT bHeightMotorEncoderHomed OR rtEncoderHomed.Q THEN
	bHeightMotorUp:=(*TRUE*) NOT tofHeightMotorDown.Q;;
	bHeightMotorDown:=FALSE;
	IF tonHeightNoChange.Q THEN
		bHeightMotorEncoderCounterReset:=TRUE;
		bHeightMotorUp:=FALSE;
	END_IF
	//Jesli enkoder zbazowany zakończ bazowanie	
	IF rtEncoderHomed.Q THEN
		bHeightMotorUp:=FALSE;
		bHeightMotorDown:=FALSE;
		eState:=E_Station.eHomingDone;
	END_IF		
		
//Po podniesieniu stacji opuszczanie do ustalonej wysokości
ELSIF bHeightMotorEncoderHomed THEN
	bHeightMotorEncoderCounterReset:=FALSE;
	bHeightMotorUp:=lrHeightMotorCV<=nPositionHeightSV;
	bHeightMotorDown:=lrHeightMotorCV>=nPositionHeightSV (*AND lrHeightMotorCV>=lrMinHeight*);
	//Kiedy stacja osiągnie wysokość zadaną
	IF ABS(lrHeightMotorCV-nPositionHeightSV)<1 OR tonLimitPosMaxReachedDelay.Q OR tonLimitPosMinReachedDelay.Q (*OR lrHeightMotorCV>=lrMinHeight*) THEN
		bHeightMotorDown:=FALSE;
		bHeightMotorUp:=FALSE;
		eState:=E_Station.eHomingDone;
	END_IF			
END_IF

	
//Opcja braku podnośnika	
IF bNoLifter THEN
	eState:=E_Station.eHomingDone;
END_IF
END_ACTION

ACTION ManualMovements:

//W trybie ruchów manualnych wykonuj ruchy za pomocą rozkazów manualnych
IF NOT bRun THEN
	bCatchActuator:=bManualCatchActuator;
	bHeightMotorUp:=bManualHeightMotorUp;
	bHeightMotorDown:=bManualHeightMotorDown;
ELSE	//Kasuje zeby po cyklu nic sie nie poruszało
	bManualCatchActuator := FALSE;
	bManualHeightMotorUp  := FALSE;
	bManualHeightMotorDown  := FALSE;
END_IF


IF bHoming OR bHeightSet THEN
	eState:=E_Station.eHoming;
END_IF
	
Running();
	
//Zabezpieczenie przed kolizją stacji poprzez ruch podnośnika	
IF bHeightMotorDown AND lrHeightMotorCV<=lrMinHeight AND NOT bHoming AND NOT bHeightSet THEN
	bHeightMotorDown:=FALSE;
END_IF	

IF bHeightMotorUp AND lrHeightMotorCV>=lrMaxHeight AND NOT bHoming AND NOT bHeightSet THEN
	bHeightMotorUp:=FALSE;
END_IF		 

IF NOT bRun THEN
	bCycleDone 					:= FALSE;
	bCycleNotDone 				:= FALSE;	
END_IF
END_ACTION

ACTION Running:

//Timery
tonCatchingTime(IN:=(eRunningState=E_CatchStationState.eCatching), PT:=T#500MS);


CASE eRunningState OF
	
	//NIEGOTOWY
	E_CatchStationState.eDisabled:
		eRunningState:=E_CatchStationState.eReady;

	//Chwytak gotowy do pracy
	E_CatchStationState.eReady: 
		//Jeśli komenda chwytania przejdz do stanu chwytanie
		IF NOT bCycleDone AND NOT bCycleNotDone THEN
			IF bRun THEN
			eRunningState:=E_CatchStationState.eCatching;
			END_IF
		END_IF
		
	//Chwytanie 
	E_CatchStationState.eCatching:
		bCatchActuator:=TRUE;
		

		IF tonCatchingTime.Q THEN
			IF bClosedActuatorSensor THEN
				eRunningState	:= E_CatchStationState.eCatched;
			ELSE
				eRunningState	:= E_CatchStationState.eNotCatched;
			END_IF
		END_IF

	//Uchwycone 
	E_CatchStationState.eCatched:
		bCatchActuator:=bRun;
		bCycleDone := TRUE;
		//Kiedy zniknie rozkaz chwytania i 
	
	E_CatchStationState.eNotCatched:
	
		bCatchActuator:=bRun;                                   
		bCycleDone := TRUE;
	
END_CASE
END_ACTION

ACTION Statistics:



rtrigCycleTimerRead(CLK:=eRunningState=E_CatchStationState.eCatched);
IF rtrigCycleTimerRead.Q THEN
	tCycleTime:=tonCycleTimer.ET;
END_IF
tonCycleTimer(IN:=eState>E_Station.eReady,PT:=T#1D);
END_ACTION

END_FUNCTION_BLOCK

// ---- POUs/P14_BadBottleConyevor.TcPOU
(*
Nazwa:			P14_BadBottleConyevor
Opis:			Stacja taśmociągu odrzuconych butelek
Wersja:			v0.1
Data:			2018-10-10
Autor:			DP
Urzadzenia:		
Konfiguracja:	
Info:

*)
PROGRAM P14_BadBottleConyevor
VAR_INPUT
	IbBadBottleConveyorFullSensor AT %I*: BOOL;			(*PLC.G1 robot*)	// Czujnik przepelnienia odrzuconych butelek
END_VAR
VAR
	
	(*****************TRANSPORTER ODRZUCONYCH BUTELEK*******************)
	//fbBadBottleConveyor							: FB_LenzeInverter;
	fbBadBottleConveyor								: FB_MitsubishiInverter;
	eBadBottleConveyorState							: E_Station;			
	eBadBottleConveyorRunningState					: E_ConveyorState;	
	fbBadBottleConveyorState						: FB_State;		
	QnBadBottleConveyorVelocitySV AT %Q*: UDINT; 			(*po kom*)	// Nastawa prędkości transportera
	InBadBottleConveyorVelocityCV AT %I*: UDINT;			(*po kom*)
	InBadBottleConveyorSTW AT %I*: UINT; 				(*po kom*)	// Statusword transportera wejściowo wyjściowego
	QnBadBottleConveyorConvCTW AT %Q*: UINT;  			(*po kom*)	// Controlword transportera we/wy
	InBadBottleConveyorErrorCode AT %I*:UINT;			(*po kom*)
	
	TimerBadBottleConveyorFullSensorWarning: TON;
	TimerBadBottleConveyorFullSensorError: TON;
	
	(*Dodatkowe ostrzezenie*)
	rtIbBadBottleConveyorFullSensor: R_TRIG;
	iBadBottleConveyorFullCounter: INT;
	tonNotIbBadBottleConveyorFullSensor: TON;
	(*Smieci*)
	bConveyorTest1											: BOOL;
	
	
	(*inne*)
	

	bTestRun: BOOL;
END_VAR

aBadBottleConveyor();

// Konwersja do wyświetlania prędkości
IF NOT VIS.bBadBottleConveyorManualDirection AND (bBadBottleConveyorStart OR VIS.bBadBottleConveyorManualCmdStart) THEN
	VIS.nBadBottleConveyorCV := 65535-InBadBottleConveyorVelocityCV;
ELSE 
	VIS.nBadBottleConveyorCV := InBadBottleConveyorVelocityCV;
END_IF





(********* GENEROWANIE STANU STACJI DO WIZKI**********)
fbBadBottleConveyorState(
	eState														:= eBadBottleConveyorState , 
	bRun														:= bBadBottleConveyorStart OR VIS.bBadBottleConveyorManualCmdStart ,	
	eConveyorRunningState										:= eBadBottleConveyorRunningState, 
	sStateDesc													=> VIS.sBadBottleConveyorState,
	iState														=> VIS.iBadBottleConveyorState	);
(***** KONIEC GENEROWANIE STANU STACJI DO WIZKI*******)

(****Ostrzezenia***)
rtIbBadBottleConveyorFullSensor(CLK:=IbBadBottleConveyorFullSensor AND P00_PackML.fbPMLAuto.ePMLState = E_PMLState.ePMLState_EXECUTE, Q=>);
IF rtIbBadBottleConveyorFullSensor.Q THEN
	iBadBottleConveyorFullCounter	:=	iBadBottleConveyorFullCounter +	1;
END_IF
tonNotIbBadBottleConveyorFullSensor(IN:=NOT IbBadBottleConveyorFullSensor AND P00_PackML.fbPMLAuto.ePMLState = E_PMLState.ePMLState_EXECUTE, PT:=T#7S);
IF tonNotIbBadBottleConveyorFullSensor.Q THEN
	iBadBottleConveyorFullCounter := 0;
END_IF

TimerBadBottleConveyorFullSensorWarning(IN:=IbBadBottleConveyorFullSensor, PT:=T#2S);

IF TimerBadBottleConveyorFullSensorWarning.Q(* OR (iBadBottleConveyorFullCounter>=3 AND NOT (P00_PackML.fbPMLAuto.ePMLState = E_PMLState.ePMLState_IDLE)))*)AND NOT BottleTransferWarning[0].bWarning THEN
	BottleTransferWarning[0].bWarning							:= TRUE;
	BottleTransferWarning[0].udiWarningCode						:= 57;
	BottleTransferWarning[0].sDescription						:= 'Transporter | Zapełniony transporter odrzuconych opakowań';
ELSIF NOT IbBadBottleConveyorFullSensor THEN//AND BottleTransferWarning[0].bAcknowledge THEN
	BottleTransferWarning[0].bWarning							:= FALSE;
	BottleTransferWarning[0].bAcknowledge						:= FALSE;
	VIS.uliWarningAcknowledge.2 								:= FALSE;
ELSIF BottleTransferWarning[0].bAcknowledge THEN
	BottleTransferWarning[0].bAcknowledge						:= TRUE;
END_IF


(*Blad zatrzymania*)
TimerBadBottleConveyorFullSensorError(IN:=TimerBadBottleConveyorFullSensorWarning.Q, PT:=T#2S);

ACTION aBadBottleConveyor:
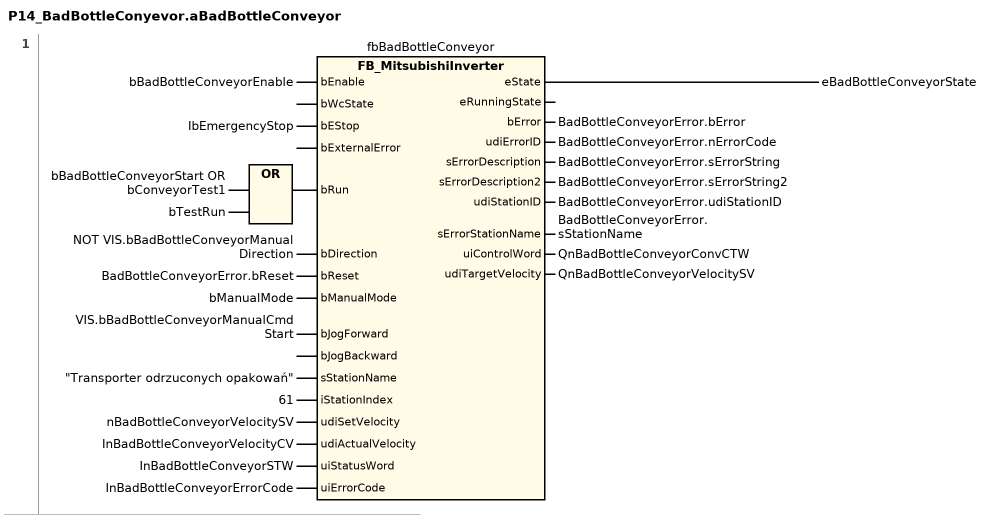
// NETWORK 1
fbBadBottleConveyor(
    bEnable := bBadBottleConveyorEnable,
    bEStop := IbEmergencyStop,
    bRun := (bBadBottleConveyorStart OR bConveyorTest1) OR bTestRun,
    bDirection := NOT VIS.bBadBottleConveyorManualDirection,
    bReset := BadBottleConveyorError.bReset,
    bManualMode := bManualMode,
    bJogForward := VIS.bBadBottleConveyorManualCmdStart,
    sStationName := "Transporter odrzuconych opakowań",
    iStationIndex := 61,
    udiSetVelocity := nBadBottleConveyorVelocitySV,
    udiActualVelocity := InBadBottleConveyorVelocityCV,
    uiStatusWord := InBadBottleConveyorSTW,
    uiErrorCode := InBadBottleConveyorErrorCode,
    bError => BadBottleConveyorError.bError,
    udiErrorID => BadBottleConveyorError.nErrorCode,
    sErrorDescription => BadBottleConveyorError.sErrorString,
    sErrorDescription2 => BadBottleConveyorError.sErrorString2,
    udiStationID => BadBottleConveyorError.udiStationID,
    sErrorStationName => BadBottleConveyorError.sStationName,
    uiControlWord => QnBadBottleConveyorConvCTW,
    udiTargetVelocity => QnBadBottleConveyorVelocitySV); // FB_MitsubishiInverter
eBadBottleConveyorState := fbBadBottleConveyor.eState;
END_ACTION

END_PROGRAM

// ---- POUs/P13_BottleTransfer.TcPOU
(*
Nazwa:			P13_BottleTransfer
Opis:			Stacja odkładania butelek w różne miejsca
Wersja:			v0.1
Data:			2018-10-10
Autor:			DP
Urzadzenia:		
Konfiguracja:	
Info:

*)
PROGRAM P13_BottleTransfer
VAR_INPUT
	IbFirstFormCheckFormSensor				AT %I*	: BOOL; 						// Sygnal pierwszej formatki
	IbSecondFormCheckFormSensor				AT %I*	: BOOL; 						// Sygnal drugiej formatki
	IbBottleCheckAfterBottleTransferSensor	AT %I*	: BOOL; 						// Wejście z czujnika wykrycia butelki za robotem
	IbBottleTransferFormAfterSensor			AT %I*: BOOL; 					// Czujnik formatki za robotem
	IbBottleTransferFormAfterSensor2			AT %I*: BOOL; 					// Czujnik 2 formatki za robotem
END_VAR
VAR
	// Blok Sterujący podajnikiem nakrętek
	fbBottleTransfer									: FB_Robot2Bottles;
	tonEnableDelay: TON;
	eBottleTransferState					: E_Station;
	eBottleTransferRunningState				: E_RobotMovState;	
	fbBottleTransferState					: FB_State;	
	
	// WEJSCIA I WYJSCIA SPRZETOWE	
	QaDataRobotIO                            AT %Q*: ARRAY[1..8] OF USINT;
    QaDataRobotREG                           AT %Q*: ARRAY[1..32] OF UINT;
    IaDataRobotIO                            AT %I*: ARRAY[1..8] OF USINT;
    IaDataRobotREG                       	 AT %I*: ARRAY[1..32] OF UINT;
	

	
	
	TimerBottleTransferEnable: TOF;
	(*Nowe od robota Mitsubishi*)
	QbBottleTransferRobotMode1 AT %Q*:BOOL; 								//Zezwalanie na pracę robota 1
	QbBottleTransferRobotMode2 AT %Q*:BOOL; 								//Zezwalanie na pracę robota 2	

//	
	
	bBottleTransferLubricationResetCase: INT;
	tonBottleTransferLubricationResetCase1: TON;
	tonBottleTransferLubricationResetCase2: TON;
	tonBottleTransferLubricationResetCase3: TON;
	tonBottleTransferLubricationResetCase4: TON;
	tonBottleTransferLubricationResetCase5: TON;
	tonBottleTransferLubricationResetCase6: TON;
	tonBottleTransferLubricationResetCase7: TON;
	bTestWarning							: BOOL;
	bTestHoming								: BOOL;
	bTestPick								: BOOL;
	bTestPlace								: BOOL;
END_VAR

IF VIS.iBottleTransferPickOffsetZShow > 40	THEN
	VIS.iBottleTransferPickOffsetZShow								:= 40;
END_IF
IF VIS.iBottleTransferPickOffsetZShow < -60	THEN
	VIS.iBottleTransferPickOffsetZShow								:= -60;
END_IF

IF VIS.iBottleTransferPick2OffsetZShow > 40 THEN
	VIS.iBottleTransferPick2OffsetZShow								:= 40;
END_IF                                              				
IF VIS.iBottleTransferPick2OffsetZShow < -40 THEN   				
	VIS.iBottleTransferPick2OffsetZShow								:= -40;
END_IF                                              				
                                                    				
IF VIS.iBottleTransferPlace1OffsetZShow > 40 THEN   				
	VIS.iBottleTransferPlace1OffsetZShow							:= 40;
END_IF                                              				
IF VIS.iBottleTransferPlace1OffsetZShow < -60 THEN  				
	VIS.iBottleTransferPlace1OffsetZShow							:= -60;
END_IF

IF VIS.iBottleTransferPlace2OffsetZShow > 40 THEN
	VIS.iBottleTransferPlace2OffsetZShow							:= 40;
END_IF
IF VIS.iBottleTransferPlace2OffsetZShow < -80 THEN
	VIS.iBottleTransferPlace2OffsetZShow							:= -80;
END_IF

IF VIS.iBottleTransferPlace2OffsetXShow < -10 THEN
	VIS.iBottleTransferPlace2OffsetXShow							:= -10;
END_IF

IF VIS.iBottleTransferSpeedShow > 100 THEN
	VIS.iBottleTransferSpeedShow									:= 100;
END_IF
IF VIS.iBottleTransferSpeedShow < 5 THEN
	VIS.iBottleTransferSpeedShow									:= 5;
END_IF

aBottleTransfer();
aStatistics();
aManualMode();
(********* GENEROWANIE STANU STACJI DO WIZKI**********)		
fbBottleTransferState(
	eState															:= eBottleTransferState , 
	bRun															:= VIS.bBottleTransferRun,	
	eCapFeederRobotRunningState										:= eBottleTransferRunningState , 
	sStateDesc														=> VIS.sBottleTransferState,
	iState															=> VIS.iBottleTransferState	);	
(***** KONIEC GENEROWANIE STANU STACJI DO WIZKI*******)	

(*Opoznienie wyłączanie enabla*)
TimerBottleTransferEnable (IN:=bBottleTransferEnable , PT:=T#2S);

aWarning();


(**Wystawienie wyjść do robota**)

//QbBottleTransferRobotMode1											:= FALSE;
//QbBottleTransferRobotMode2											:= FALSE;

QbBottleTransferRobotMode1											:= TRUE;
QbBottleTransferRobotMode2											:= TRUE;

(**Koniec wystawienie wyjść do robota**)

ACTION aBottleTransfer:
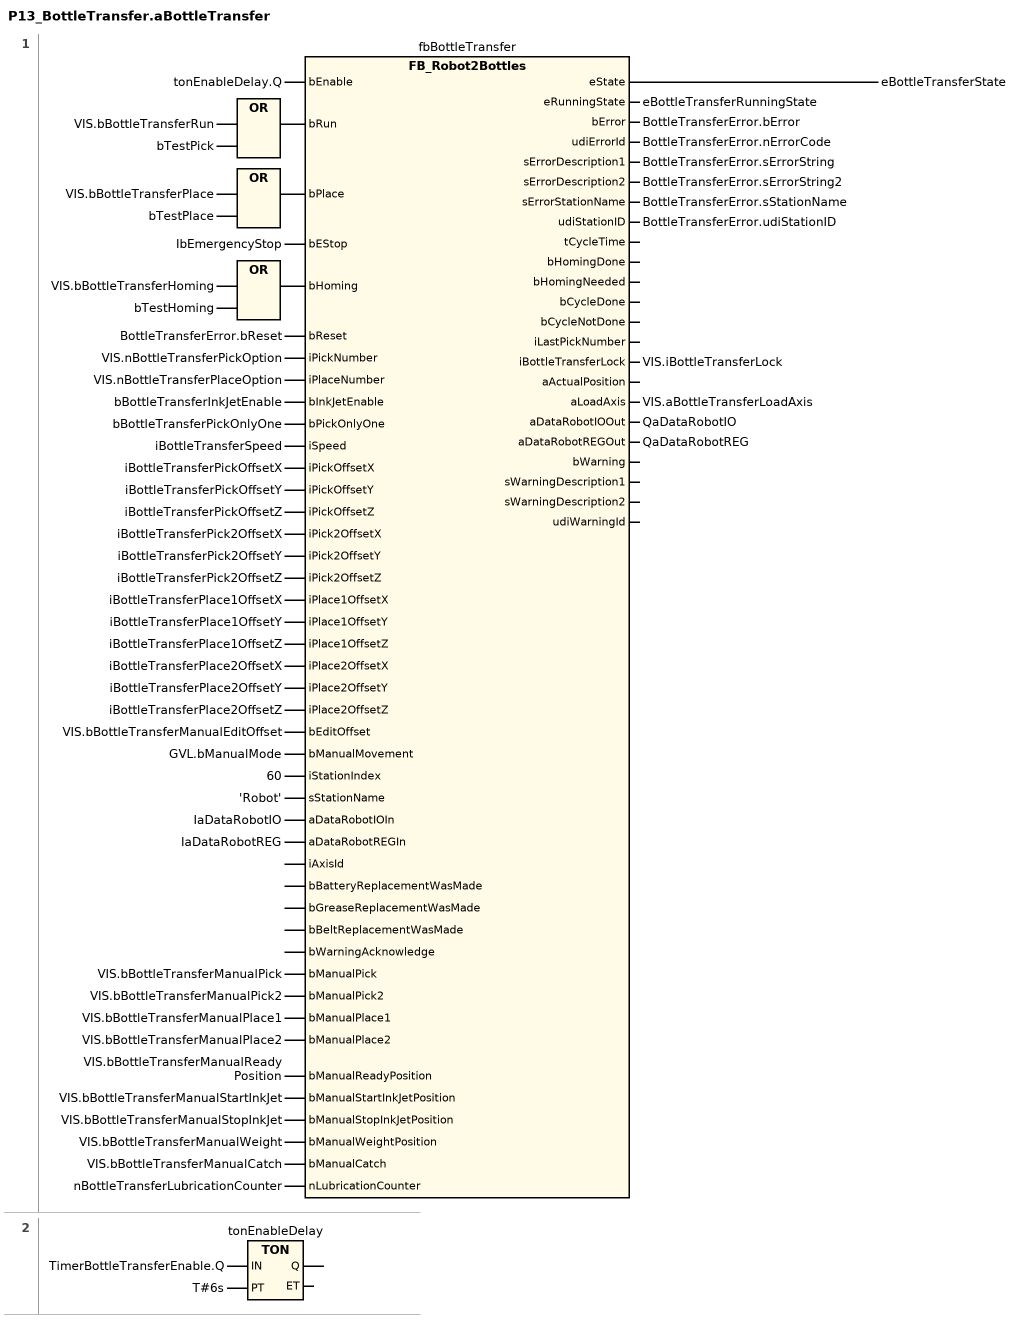
// NETWORK 1
fbBottleTransfer(
    bEnable := tonEnableDelay.Q,
    bRun := VIS.bBottleTransferRun OR bTestPick,
    bPlace := VIS.bBottleTransferPlace OR bTestPlace,
    bEStop := IbEmergencyStop,
    bHoming := VIS.bBottleTransferHoming OR bTestHoming,
    bReset := BottleTransferError.bReset,
    iPickNumber := VIS.nBottleTransferPickOption,
    iPlaceNumber := VIS.nBottleTransferPlaceOption,
    bInkJetEnable := bBottleTransferInkJetEnable,
    bPickOnlyOne := bBottleTransferPickOnlyOne,
    iSpeed := iBottleTransferSpeed,
    iPickOffsetX := iBottleTransferPickOffsetX,
    iPickOffsetY := iBottleTransferPickOffsetY,
    iPickOffsetZ := iBottleTransferPickOffsetZ,
    iPick2OffsetX := iBottleTransferPick2OffsetX,
    iPick2OffsetY := iBottleTransferPick2OffsetY,
    iPick2OffsetZ := iBottleTransferPick2OffsetZ,
    iPlace1OffsetX := iBottleTransferPlace1OffsetX,
    iPlace1OffsetY := iBottleTransferPlace1OffsetY,
    iPlace1OffsetZ := iBottleTransferPlace1OffsetZ,
    iPlace2OffsetX := iBottleTransferPlace2OffsetX,
    iPlace2OffsetY := iBottleTransferPlace2OffsetY,
    iPlace2OffsetZ := iBottleTransferPlace2OffsetZ,
    bEditOffset := VIS.bBottleTransferManualEditOffset,
    bManualMovement := GVL.bManualMode,
    iStationIndex := 60,
    sStationName := 'Robot',
    aDataRobotIOIn := IaDataRobotIO,
    aDataRobotREGIn := IaDataRobotREG,
    bManualPick := VIS.bBottleTransferManualPick,
    bManualPick2 := VIS.bBottleTransferManualPick2,
    bManualPlace1 := VIS.bBottleTransferManualPlace1,
    bManualPlace2 := VIS.bBottleTransferManualPlace2,
    bManualReadyPosition := VIS.bBottleTransferManualReadyPosition,
    bManualStartInkJetPosition := VIS.bBottleTransferManualStartInkJet,
    bManualStopInkJetPosition := VIS.bBottleTransferManualStopInkJet,
    bManualWeightPosition := VIS.bBottleTransferManualWeight,
    bManualCatch := VIS.bBottleTransferManualCatch,
    nLubricationCounter := nBottleTransferLubricationCounter,
    eRunningState => eBottleTransferRunningState,
    bError => BottleTransferError.bError,
    udiErrorId => BottleTransferError.nErrorCode,
    sErrorDescription1 => BottleTransferError.sErrorString,
    sErrorDescription2 => BottleTransferError.sErrorString2,
    sErrorStationName => BottleTransferError.sStationName,
    udiStationID => BottleTransferError.udiStationID,
    iBottleTransferLock => VIS.iBottleTransferLock,
    aLoadAxis => VIS.aBottleTransferLoadAxis,
    aDataRobotIOOut => QaDataRobotIO,
    aDataRobotREGOut => QaDataRobotREG); // FB_Robot2Bottles
eBottleTransferState := fbBottleTransfer.eState;

// NETWORK 2
tonEnableDelay(IN := TimerBottleTransferEnable.Q, PT := T#6s); // TON
END_ACTION

ACTION aManualMode:
	//iBottleTransferLock									:INT;					// Blokowanie przycisków trybu manualnego (b0-1 blokuj 
																					// 2#11111111 - nie moge nic  
																					// 2#11111110 - moge pobrać (tylko Pick1 i Pick 2 odblokowane)
																					// 2#11101001 - moge odłożyć, odrzucić i pojechać przed inkjet		
																					// 2#11110111 - moge jechać tylko do gotowości
																					// 2#11110111 - moge jechać tylko do gotowości
																					// 2#11011111 - moge jechać do koniec inkjet
																					// 2#10101101 - moge odłożyć na ety., wrocić przed inkjet
																					// 2#11111110 - moge pobrać
IF	 VIS.iBottleTransferLock = 2#11111111 THEN //2#11111111 - nie moge nic  
		VIS.bBottleTransferManualCatchVisibility				:= FALSE;					 	// Chwytak - przycisk odblokowany
  	  	VIS.bBottleTransferManualPickVisibility					:= FALSE; 						// Pobierz 1 but. - przycisk odblokowany
		VIS.bBottleTransferManualPick2Visibility 				:= FALSE; 						// Pobierz 2 but. - przycisk odblokowany
  	 	VIS.bBottleTransferManualPlace1Visibility				:= FALSE; 						// Odłóż na etykieciarkę - przycisk odblokowany
  	 	VIS.bBottleTransferManualPlace2Visibility				:= FALSE; 						// Odłóż na odrzut - przycisk odblokowany
  	 	VIS.bBottleTransferManualReadyPositionVisibility		:= FALSE; 						// Gotowość - przycisk odblokowany
		VIS.bBottleTransferManualStartInkJetVisibility			:= FALSE; 						// Start InkJet - przycisk odblokowany
		VIS.bBottleTransferManualStopInkJetVisibility			:= FALSE; 						// Stop InkJet - przycisk odblokowany	
ELSIF VIS.iBottleTransferLock = 2#11111110 THEN //2#11111110 - moge pobrać (tylko Pick1 i Pick 2 odblokowane)  
		VIS.bBottleTransferManualCatchVisibility				:= FALSE;					 	// Chwytak - przycisk odblokowany
  	  	VIS.bBottleTransferManualPickVisibility					:= TRUE; 						// Pobierz 1 but. - przycisk odblokowany
		VIS.bBottleTransferManualPick2Visibility 				:= TRUE;  						// Pobierz 2 but. - przycisk odblokowany
  	 	VIS.bBottleTransferManualPlace1Visibility				:= FALSE; 						// Odłóż na etykieciarkę - przycisk odblokowany
  	 	VIS.bBottleTransferManualPlace2Visibility				:= FALSE; 						// Odłóż na odrzut - przycisk odblokowany
  	 	VIS.bBottleTransferManualReadyPositionVisibility		:= FALSE; 						// Gotowość - przycisk odblokowany
		VIS.bBottleTransferManualStartInkJetVisibility			:= FALSE; 						// Start InkJet - przycisk odblokowany
		VIS.bBottleTransferManualStopInkJetVisibility			:= FALSE; 						// Stop InkJet - przycisk odblokowany		
ELSIF VIS.iBottleTransferLock = 2#11101001 THEN //2#11101001 - moge odłożyć, odrzucić i pojechać przed inkjet	
 		VIS.bBottleTransferManualCatchVisibility				:= FALSE;					 	// Chwytak - przycisk odblokowany
  	  	VIS.bBottleTransferManualPickVisibility					:= FALSE; 						// Pobierz 1 but. - przycisk odblokowany
		VIS.bBottleTransferManualPick2Visibility 				:= FALSE; 						// Pobierz 2 but. - przycisk odblokowany
  	 	VIS.bBottleTransferManualPlace1Visibility				:= TRUE; 						// Odłóż na etykieciarkę - przycisk odblokowany
  	 	VIS.bBottleTransferManualPlace2Visibility				:= TRUE;  						// Odłóż na odrzut - przycisk odblokowany
  	 	VIS.bBottleTransferManualReadyPositionVisibility		:= FALSE; 						// Gotowość - przycisk odblokowany
		VIS.bBottleTransferManualStartInkJetVisibility			:= TRUE;  						// Start InkJet - przycisk odblokowany
		VIS.bBottleTransferManualStopInkJetVisibility			:= FALSE; 						// Stop InkJet - przycisk odblokowany	
ELSIF VIS.iBottleTransferLock = 2#11110111 THEN //2#11110111 - moge jechać tylko do gotowości 
		VIS.bBottleTransferManualCatchVisibility				:= FALSE;					 	// Chwytak - przycisk odblokowany
  	  	VIS.bBottleTransferManualPickVisibility					:= FALSE; 						// Pobierz 1 but. - przycisk odblokowany
		VIS.bBottleTransferManualPick2Visibility 				:= FALSE; 						// Pobierz 2 but. - przycisk odblokowany
  	 	VIS.bBottleTransferManualPlace1Visibility				:= FALSE; 						// Odłóż na etykieciarkę - przycisk odblokowany
  	 	VIS.bBottleTransferManualPlace2Visibility				:= FALSE; 						// Odłóż na odrzut - przycisk odblokowany
  	 	VIS.bBottleTransferManualReadyPositionVisibility		:= TRUE; 						// Gotowość - przycisk odblokowany
		VIS.bBottleTransferManualStartInkJetVisibility			:= FALSE; 						// Start InkJet - przycisk odblokowany
		VIS.bBottleTransferManualStopInkJetVisibility			:= FALSE; 						// Stop InkJet - przycisk odblokowany	
ELSIF VIS.iBottleTransferLock = 2#11110111 THEN //2#11110111 - moge jechać tylko do gotowości 
		VIS.bBottleTransferManualCatchVisibility				:= FALSE;					 	// Chwytak - przycisk odblokowany
  	  	VIS.bBottleTransferManualPickVisibility					:= FALSE; 						// Pobierz 1 but. - przycisk odblokowany
		VIS.bBottleTransferManualPick2Visibility 				:= FALSE; 						// Pobierz 2 but. - przycisk odblokowany
  	 	VIS.bBottleTransferManualPlace1Visibility				:= FALSE; 						// Odłóż na etykieciarkę - przycisk odblokowany
  	 	VIS.bBottleTransferManualPlace2Visibility				:= FALSE; 						// Odłóż na odrzut - przycisk odblokowany
  	 	VIS.bBottleTransferManualReadyPositionVisibility		:= TRUE;  						// Gotowość - przycisk odblokowany
		VIS.bBottleTransferManualStartInkJetVisibility			:= FALSE; 						// Start InkJet - przycisk odblokowany
		VIS.bBottleTransferManualStopInkJetVisibility			:= FALSE; 						// Stop InkJet - przycisk odblokowany	
ELSIF VIS.iBottleTransferLock = 2#11011111 THEN //2#11011111 - moge jechać do koniec inkjet  
		VIS.bBottleTransferManualCatchVisibility				:= FALSE;					 	// Chwytak - przycisk odblokowany
  	  	VIS.bBottleTransferManualPickVisibility					:= FALSE; 						// Pobierz 1 but. - przycisk odblokowany
		VIS.bBottleTransferManualPick2Visibility 				:= FALSE; 						// Pobierz 2 but. - przycisk odblokowany
  	 	VIS.bBottleTransferManualPlace1Visibility				:= FALSE; 						// Odłóż na etykieciarkę - przycisk odblokowany
  	 	VIS.bBottleTransferManualPlace2Visibility				:= FALSE; 						// Odłóż na odrzut - przycisk odblokowany
  	 	VIS.bBottleTransferManualReadyPositionVisibility		:= FALSE; 						// Gotowość - przycisk odblokowany
		VIS.bBottleTransferManualStartInkJetVisibility			:= FALSE; 						// Start InkJet - przycisk odblokowany
		VIS.bBottleTransferManualStopInkJetVisibility			:= TRUE;  						// Stop InkJet - przycisk odblokowany	
ELSIF VIS.iBottleTransferLock = 2#10101101 THEN //2#10101101 - moge odłożyć na ety., wrocić przed inkjet  
		VIS.bBottleTransferManualCatchVisibility				:= FALSE;					 	// Chwytak - przycisk odblokowany
  	  	VIS.bBottleTransferManualPickVisibility					:= FALSE; 						// Pobierz 1 but. - przycisk odblokowany
		VIS.bBottleTransferManualPick2Visibility 				:= FALSE; 						// Pobierz 2 but. - przycisk odblokowany
  	 	VIS.bBottleTransferManualPlace1Visibility				:= TRUE;  						// Odłóż na etykieciarkę - przycisk odblokowany
  	 	VIS.bBottleTransferManualPlace2Visibility				:= FALSE; 						// Odłóż na odrzut - przycisk odblokowany
  	 	VIS.bBottleTransferManualReadyPositionVisibility		:= FALSE; 						// Gotowość - przycisk odblokowany
		VIS.bBottleTransferManualStartInkJetVisibility			:= TRUE;  						// Start InkJet - przycisk odblokowany
		VIS.bBottleTransferManualStopInkJetVisibility			:= FALSE; 						// Stop InkJet - przycisk odblokowany	
ELSIF VIS.iBottleTransferLock = 2#11111110 THEN //2#11111110 - moge pobrać 	
		VIS.bBottleTransferManualCatchVisibility				:= FALSE;					 	// Chwytak - przycisk odblokowany
  	  	VIS.bBottleTransferManualPickVisibility					:= TRUE;						// Pobierz 1 but. - przycisk odblokowany
		VIS.bBottleTransferManualPick2Visibility 				:= FALSE; 						// Pobierz 2 but. - przycisk odblokowany
  	 	VIS.bBottleTransferManualPlace1Visibility				:= FALSE; 						// Odłóż na etykieciarkę - przycisk odblokowany
  	 	VIS.bBottleTransferManualPlace2Visibility				:= FALSE; 						// Odłóż na odrzut - przycisk odblokowany
  	 	VIS.bBottleTransferManualReadyPositionVisibility		:= FALSE; 						// Gotowość - przycisk odblokowany
		VIS.bBottleTransferManualStartInkJetVisibility			:= FALSE; 						// Start InkJet - przycisk odblokowany
		VIS.bBottleTransferManualStopInkJetVisibility			:= FALSE; 						// Stop InkJet - przycisk odblokowany	
END_IF
END_ACTION

ACTION aStatistics:
VIS.iBottleTransferState				;
VIS.sBottleTransferState				;
VIS.bBottleTransferHoming				;
VIS.bBottleTransferHeightSet 			;
VIS.bBottleTransferIgnoreErrors			;
VIS.bBottleTransferRun					;
VIS.bBottleTransferPlace				;
VIS.nBottleTransferPlaceOption			;
VIS.nBottleTransferPickOption			;
VIS.bBottleTransferManualCatch			;
VIS.bBottleTransferManualPick			;
VIS.bBottleTransferManualPick2 			;
VIS.bBottleTransferManualPlace1			;
VIS.bBottleTransferManualPlace2			;
VIS.bBottleTransferManualReadyPosition	;
VIS.bBottleTransferManualStartInkJet	;
VIS.bBottleTransferManualStopInkJet		;
VIS.bBottleTransferManualEditOffset		;
VIS.bBottleTransferAllFormsToLabeler	;
VIS.bBottleTransferAllFormsToExit		;
VIS.bBottleTransferLubricationReset		;
VIS.aBottleTransferLoadAxis				;
VIS.iBottleTransferLock					;
END_ACTION

ACTION aWarning:
(****Ostrzezenia***)

//BottleTransferWarning[1].sDescription								:= 'Przeprowadzić smarowanie i przegląd techniczny robota';
BottleTransferWarning[1].sDescription								:= fbBottleTransfer.sWarningDescription1;
IF BottleTransferWarning[1].sDescription = '' THEN
	BottleTransferWarning[1].sDescription := 'Robot | Ostrzeżenie';
END_IF
//IF nBottleTransferLubricationCounter>900000 AND NOT BottleTransferWarning[1].bWarning THEN

tonBottleTransferLubricationResetCase1 	(IN:=bBottleTransferLubricationResetCase=10 OR bBottleTransferLubricationResetCase=300, PT:=T#1S);
tonBottleTransferLubricationResetCase2 	(IN:=bBottleTransferLubricationResetCase=100 OR bBottleTransferLubricationResetCase=200, PT:=T#1S);
tonBottleTransferLubricationResetCase3 	(IN:=bBottleTransferLubricationResetCase=110 OR bBottleTransferLubricationResetCase=210, PT:=T#1S);
tonBottleTransferLubricationResetCase4 	(IN:=bBottleTransferLubricationResetCase=120 OR bBottleTransferLubricationResetCase=220, PT:=T#1S);
tonBottleTransferLubricationResetCase5 	(IN:=bBottleTransferLubricationResetCase=130 OR bBottleTransferLubricationResetCase=230, PT:=T#1S);
tonBottleTransferLubricationResetCase6 	(IN:=bBottleTransferLubricationResetCase=140 OR bBottleTransferLubricationResetCase=240, PT:=T#1S);
tonBottleTransferLubricationResetCase7 	(IN:=bBottleTransferLubricationResetCase=150 OR bBottleTransferLubricationResetCase=250, PT:=T#1S);

IF (fbBottleTransfer.bWarning OR bTestWarning) AND NOT BottleTransferWarning[1].bWarning THEN
	BottleTransferWarning[1].bWarning								:= TRUE;
	BottleTransferWarning[1].udiWarningCode							:= 58;
ELSIF BottleTransferWarning[1].bAcknowledge THEN
	
	CASE bBottleTransferLubricationResetCase OF 
		
		0:
			fbBottleTransfer.iAxisId					:= 0 ;
			fbBottleTransfer.bBatteryReplacementWasMade	:= FALSE;			
			fbBottleTransfer.bGreaseReplacementWasMade	:= FALSE;		
			fbBottleTransfer.bBeltReplacementWasMade	:= FALSE;		
			fbBottleTransfer.bWarningAcknowledge		:= FALSE;		

			//battery
			//1330,0111,7450,7451,7510,7520			
			//grease
			//7121,7122,7123,7124,7125,7126,7530			
			//belt
			//7131,7132,7133,7134,7135,7136,7540
			
			IF	//baterry 
				fbBottleTransfer.udiWarningId =	1330 OR fbBottleTransfer.udiWarningId =	0111 OR	
				fbBottleTransfer.udiWarningId =	7450 OR fbBottleTransfer.udiWarningId =	7451 OR
				fbBottleTransfer.udiWarningId =	7510 OR fbBottleTransfer.udiWarningId =	7520 		
				THEN
				bBottleTransferLubricationResetCase	:=	10;
			ELSIF	//grease
				fbBottleTransfer.udiWarningId =	7121 OR fbBottleTransfer.udiWarningId =	7122 OR	
				fbBottleTransfer.udiWarningId =	7123 OR fbBottleTransfer.udiWarningId =	7124 OR
				fbBottleTransfer.udiWarningId =	7125 OR fbBottleTransfer.udiWarningId =	7126 OR
				fbBottleTransfer.udiWarningId =	7530 
				THEN
				bBottleTransferLubricationResetCase	:=	100;
			ELSIF	//belt
				fbBottleTransfer.udiWarningId =	7131 OR fbBottleTransfer.udiWarningId =	7132 OR	
				fbBottleTransfer.udiWarningId =	7133 OR fbBottleTransfer.udiWarningId =	7134 OR
				fbBottleTransfer.udiWarningId =	7135 OR fbBottleTransfer.udiWarningId =	7136 OR
				fbBottleTransfer.udiWarningId =	7540 
				THEN
				bBottleTransferLubricationResetCase	:=	200;
			ELSE	//other
				bBottleTransferLubricationResetCase	:=	300;
						
			END_IF
			
		10: //battery
			fbBottleTransfer.bBatteryReplacementWasMade	:=	TRUE;			
			fbBottleTransfer.bWarningAcknowledge		:=	TRUE;
			IF tonBottleTransferLubricationResetCase1.Q THEN
				bBottleTransferLubricationResetCase		:=	1000;
			END_IF
		
		100: //grease
			fbBottleTransfer.iAxisId					:= 1 ;	
			fbBottleTransfer.bGreaseReplacementWasMade	:= TRUE;		
			fbBottleTransfer.bWarningAcknowledge		:= TRUE;
			IF tonBottleTransferLubricationResetCase2.Q THEN
				bBottleTransferLubricationResetCase		:=	bBottleTransferLubricationResetCase	+	10;
			END_IF
		110://grease
			fbBottleTransfer.iAxisId					:= 2 ;	
			fbBottleTransfer.bGreaseReplacementWasMade	:= TRUE;		
			fbBottleTransfer.bWarningAcknowledge		:= TRUE;
			IF tonBottleTransferLubricationResetCase3.Q THEN
				bBottleTransferLubricationResetCase		:=	bBottleTransferLubricationResetCase	+	10;
			END_IF			
		120: //grease
			fbBottleTransfer.iAxisId					:= 3 ;	
			fbBottleTransfer.bGreaseReplacementWasMade	:= TRUE;		
			fbBottleTransfer.bWarningAcknowledge		:= TRUE;
			IF tonBottleTransferLubricationResetCase4.Q THEN
				bBottleTransferLubricationResetCase		:=	bBottleTransferLubricationResetCase	+	10;
			END_IF	
		130://grease
			fbBottleTransfer.iAxisId					:= 4 ;	
			fbBottleTransfer.bGreaseReplacementWasMade	:= TRUE;		
			fbBottleTransfer.bWarningAcknowledge		:= TRUE;
			IF tonBottleTransferLubricationResetCase5.Q THEN
				bBottleTransferLubricationResetCase		:=	bBottleTransferLubricationResetCase	+	10;
			END_IF	
		140://grease
			fbBottleTransfer.iAxisId					:= 5 ;	
			fbBottleTransfer.bGreaseReplacementWasMade	:= TRUE;		
			fbBottleTransfer.bWarningAcknowledge		:= TRUE;
			IF tonBottleTransferLubricationResetCase6.Q THEN
				bBottleTransferLubricationResetCase		:=	bBottleTransferLubricationResetCase	+	10;
			END_IF	
		150://grease
			fbBottleTransfer.iAxisId					:= 6 ;	
			fbBottleTransfer.bGreaseReplacementWasMade	:= TRUE;		
			fbBottleTransfer.bWarningAcknowledge		:= TRUE;
			IF tonBottleTransferLubricationResetCase7.Q THEN
				bBottleTransferLubricationResetCase		:=	1000;;
			END_IF				
			
		200: //belt
			fbBottleTransfer.iAxisId					:= 1 ;	
			fbBottleTransfer.bBeltReplacementWasMade	:= TRUE;		
			fbBottleTransfer.bWarningAcknowledge		:= TRUE;		
			IF tonBottleTransferLubricationResetCase2.Q  THEN
				bBottleTransferLubricationResetCase		:=	bBottleTransferLubricationResetCase	+	10;
			END_IF
		210: //belt
			fbBottleTransfer.iAxisId					:= 2 ;	
			fbBottleTransfer.bBeltReplacementWasMade	:= TRUE;		
			fbBottleTransfer.bWarningAcknowledge		:= TRUE;		
			IF tonBottleTransferLubricationResetCase3.Q THEN
				bBottleTransferLubricationResetCase		:=	bBottleTransferLubricationResetCase	+	10;
			END_IF		
		220: //belt
			fbBottleTransfer.iAxisId					:= 3 ;	
			fbBottleTransfer.bBeltReplacementWasMade	:= TRUE;		
			fbBottleTransfer.bWarningAcknowledge		:= TRUE;		
			IF (*tonBottleTransferLubricationResetCase4.Q*) fbBottleTransfer.bBeltReplenishmentFinished THEN
				bBottleTransferLubricationResetCase		:=	bBottleTransferLubricationResetCase	+	10;
			END_IF	
		230: //belt
			fbBottleTransfer.iAxisId					:= 4 ;	
			fbBottleTransfer.bBeltReplacementWasMade	:= TRUE;		
			fbBottleTransfer.bWarningAcknowledge		:= TRUE;		
			IF (*tonBottleTransferLubricationResetCase5.Q*) fbBottleTransfer.bBeltReplenishmentFinished THEN
				bBottleTransferLubricationResetCase		:=	bBottleTransferLubricationResetCase	+	10;
			END_IF	
		240: //belt
			fbBottleTransfer.iAxisId					:= 5;	
			fbBottleTransfer.bBeltReplacementWasMade	:= TRUE;		
			fbBottleTransfer.bWarningAcknowledge		:= TRUE;		
			IF tonBottleTransferLubricationResetCase6.Q THEN
				bBottleTransferLubricationResetCase		:=	bBottleTransferLubricationResetCase	+	10;
			END_IF	
		250: //belt
			fbBottleTransfer.iAxisId					:= 6 ;	
			fbBottleTransfer.bBeltReplacementWasMade	:= TRUE;		
			fbBottleTransfer.bWarningAcknowledge		:= TRUE;		
			IF tonBottleTransferLubricationResetCase7.Q THEN
				bBottleTransferLubricationResetCase		:=	1000;
			END_IF	
			
		300://Other		
			fbBottleTransfer.bWarningAcknowledge		:=	TRUE;
			IF tonBottleTransferLubricationResetCase1.Q THEN
				bBottleTransferLubricationResetCase		:=	1000;
			END_IF
		
		1000: //end
		
			fbBottleTransfer.iAxisId					:= 0 ;
			fbBottleTransfer.bBatteryReplacementWasMade	:= FALSE;			
			fbBottleTransfer.bGreaseReplacementWasMade	:= FALSE;		
			fbBottleTransfer.bBeltReplacementWasMade	:= FALSE;		
			fbBottleTransfer.bWarningAcknowledge		:= FALSE;	
		
			bBottleTransferLubricationResetCase								:= 0;
			BottleTransferWarning[1].bWarning								:= FALSE;
			BottleTransferWarning[1].bAcknowledge							:= FALSE;
			VIS.uliWarningAcknowledge.5 										:= FALSE;
			//nBottleTransferLubricationCounter 								:= 0;
			VIS.bBottleTransferLubricationReset 							:= FALSE;
	
	END_CASE
	


	
END_IF
END_ACTION

END_PROGRAM

// ---- POUs/FB/FB_Robot2Bottles.TcPOU
(*
Nazwa:			FB_Robot2Bottles
Opis:			Robot podwójny
Wersja:			v0.91
Data:			2025-09-04
Autor:			TW,DP
Urzadzenia:		Mistsubishi
Konfiguracja:	
Zmiany:
- 20250904 [DP] EventLog-do sprawdzenia, 1 spr->wywołać błędy 
- 20241129 [DP] ReadyPlace w aborted, bRunProgramRC Aborted->Manual
Info: 

*)
FUNCTION_BLOCK FB_Robot2Bottles
VAR_INPUT
	bEnable									: BOOL;
	bRun									: BOOL;
	bPlace									: BOOL;
	bEStop									: BOOL;
	bHoming									: BOOL;
	bReset									: BOOL;
	iPickNumber								: INT;
	iPlaceNumber							: INT;
	bInkJetEnable							: BOOL;
	bPickOnlyOne							: BOOL; {warning 'Dorobić opcje pobierania tylko jednego opakowania, jeżeli będzie taka potrzeba'}
	iSpeed									: INT;
	iPickOffsetX							: INT;
	iPickOffsetY							: INT;  
	iPickOffsetZ							: INT; 
	iPick2OffsetX							: INT;
	iPick2OffsetY							: INT;  
	iPick2OffsetZ							: INT; 
	iPlace1OffsetX							: INT;
	iPlace1OffsetY							: INT;  
	iPlace1OffsetZ							: INT;
	iPlace2OffsetX							: INT;
	iPlace2OffsetY							: INT;
	iPlace2OffsetZ							: INT; 
	bEditOffset								: BOOL;		
	bManualMovement							: BOOL;
	iStationIndex							: UDINT;					
	sStationName							: STRING;		
	aDataRobotIOIn							: ARRAY[1..8] OF USINT;
	aDataRobotREGIn							: ARRAY[1..32] OF UINT;
	
	iCaseReset								: INT;
	
	iAxisId									: INT;	
	bBatteryReplacementWasMade				: BOOL;
	bGreaseReplacementWasMade				: BOOL;
	bBeltReplacementWasMade					: BOOL;
	bWarningAcknowledge						: BOOL;




END_VAR

VAR_OUTPUT
	
	eState									: E_Station;						//Stan ogólny bloku
	eRunningState							: E_RobotMovState;					//Stan podbloku
	bError									: BOOL;								//Błąd stacji
	udiErrorId								: UDINT;							//Nr błędu grzałki zasadniczej
	sErrorDescription1						: STRING(200);							//Opis błędu
	sErrorDescription2						: STRING(200);							//Opis błędu
	sErrorStationName						: STRING;							//Nazwa stacji
	udiStationID							: UDINT;							// Nr stacji

	tCycleTime								: TIME;	
	bHomingDone								: BOOL;								//Bazowanie wykonane
	bHomingNeeded 							: BOOL;								
	bCycleDone								: BOOL;
	bCycleNotDone							: BOOL;
	iLastPickNumber							: INT;
	iBottleTransferLock						: INT;
	aActualPosition							: ARRAY[0..3] OF INT;
	aLoadAxis								: ARRAY[0..3] OF INT;
	aDataRobotIOOut							: ARRAY[1..8] OF USINT;
	aDataRobotREGOut						: ARRAY[1..32] OF UINT;
	bWarning								: BOOL;
	sWarningDescription1					: STRING;
	sWarningDescription2					: STRING;
	udiWarningId							: UDINT;
	
	
END_VAR

VAR_IN_OUT
	
	bManualPick								: BOOL;
	bManualPick2							: BOOL;
	bManualPlace1							: BOOL;
	bManualPlace2							: BOOL;
	bManualReadyPosition					: BOOL;
	bManualStartInkJetPosition				: BOOL;
	bManualStopInkJetPosition				: BOOL;
	bManualWeightPosition					: BOOL;
	bManualCatch							: BOOL;
	nLubricationCounter						: DINT;	//Licznik czasu samrowania
END_VAR

VAR
	iCaseRC									: INT;
	iLastCaseRC								: INT;
	iActualCase								: INT;	
	iCaseInit								: INT;
	iCaseHoming								: INT;
	iCaseManual								: INT;
	iTemperatureRC							: INT;
	bReadyRC								: BOOL;
	bSafePositionRC							: BOOL;
	bResetErrorRC							: BOOL;
	bErrorRCActive							: BOOL;
	bServoONRC								: BOOL;
	bServoONRCActive						: BOOL;
	bServoOFFRC								: BOOL;
	bServoOFFRCActive						: BOOL;
	bOperationEnableRC						: BOOL;
	bOperationEnableRCActive				: BOOL;
	bErrorNumberRequest						: BOOL;
	bRunProgramRC							: BOOL;
	bRunProgramRCActive						: BOOL;
	bProgramResetRC							: BOOL;
	bProgramSelectRCActive					: BOOL;
	bCatcherCloseSensor						: BOOL;
	bComingUp								: BOOL;
	bSlowMotion								: BOOL;
	IODATA									: UDINT;
	ftCapFeederRobotEditOffset				: F_TRIG;
	rtCapFeederRobotEditOffset				: R_TRIG;
	tonRetryInit							: TON;	
	tonErrorDelay							: TON;	
	tonReadyError							: TON;
	iErrorCase								: INT;
	iSpeedSend								: INT;

	tonWaitForSuckerSensor					: TON;
	iZ										: INT;
	rtPick									: R_TRIG;
	
	iActualLastCase							: INT;
	aDataRobotIn							: INT;
	rtrigCycleTimerRead						: R_TRIG;
	tonCycleTimer							: TON;
	bLowLevelErrorRCActive					: BOOL;
	bWarningRCActive						: BOOL;
	bBatteryLowVoltage						: BOOL;
	bBatteryReplenishmentFinished			: BOOL;
	bGreaseReplenishmentFinished			: BOOL;
	bBeltReplenishmentFinished				: BOOL;
	tonbStateError							: TON;
	bStateError								: BOOL;
	udiHighLevelErrorId						: UDINT;
	udiMaintenanceErrorId					: UDINT;
	udiLowLevelErrorId						: UDINT;
	rtPlace									: R_TRIG;
	bHighLevelErrorRCActive					: BOOL;
	bErrorNumberRequestActive				: BOOL;
	
	fbIntTo2Byte							: FB_IntTo2Byte;
	IODATATest								: UDINT;
// dane wysyłane liczbowo do robota	
	udiIoDATARCWrite						: UDINT;	
	
	
// Wymiana smaru i paskow	
// Sygnaly wystawiane do robota
	bBatteryReplacementDone			: BOOL;	
	bGreaseReplacementDone			: BOOL;	
	bBeltReplacementDone			: BOOL;	

	
	bBeltReplacementDoneAxis3		: BOOL;
	bBeltReplacementDoneAxis4		: BOOL;
	
	bGreaseReplacementDoneAxis1		: BOOL;	
	bGreaseReplacementDoneAxis2		: BOOL;	
	bGreaseReplacementDoneAxis3		: BOOL;	
	
	
	udiErrorIdInit: UDINT;
	bWarningNumberRequest: BOOL;

	bResetWarningRC: BOOL;
	
	
		//Zmienne od EVENTLOGGER
	bAlarmInit 						: BOOL := TRUE; 
	nAlarmNumerator					: INT;
	arfbAlarm						: ARRAY[0..19] OF  FB_TcAlarm;		//Tablica bloczków błędów
	fbSourceInfo 					: FB_TcSourceInfo;
	iSourceInfo						: I_TcSourceInfo;
	sAlarmTest						: STRING;
	//Koniec zmiennych od EVENTLOGGER
END_VAR


Control();
DataExchange();
ErrorHandling();
Warning();
LubricationCounter();
aStatistic();
aStationID();

//Zabezpieczneie przed błędem 0 dp
IF udiErrorId = 0 AND bError THEN
	udiErrorId := 311;
	//udiErrorId := 999;	
END_IF

ACTION aStationID:
udiStationID	:=	iStationIndex;
END_ACTION

ACTION aStatistic:

//Statystyka do zliczania czasu cyklu 
rtrigCycleTimerRead(CLK:=bCycleDone);


	IF rtrigCycleTimerRead.Q THEN
		tCycleTime:=tonCycleTimer.ET;
	END_IF
	
tonCycleTimer(IN:= eRunningState<>E_RobotMovState.eReadyPlace , PT:=T#1D);
END_ACTION

ACTION Control:

	iSpeedSend := iSpeed;
	
	IF iPlaceNumber = 2 THEN
		iSpeedSend := REAL_TO_INT(iSpeed / 2);
	END_IF
	
	(*****Wyłączenie enable*****)
	IF NOT bEnable THEN
		IF eState <> E_Station.eDisabled AND eState <> E_Station.ePreparingToDisable THEN
				eState 				:= E_Station.ePreparingToDisable; 
		END_IF	
	END_IF

	(*****Estop*****)
	IF NOT bEstop  THEN	
		IF eState <> E_Station.eAborted AND eState <> E_Station.eAborting AND eState <> E_Station.eDisabled THEN
				eState 				:= E_Station.eAborting; 
		END_IF
	END_IF

	
	CASE eState OF
	/////////////////////////////	
		E_Station.eDisabled: 					// Stan nieaktywnosci (Stacja wyłączona) 
		
			iCaseInit				:= 0;
			IF bEnable THEN
				eState 				:= E_Station.ePreparingToReady; 
			END_IF 
			
    /////////////////////////////	    
		E_Station.eAborted: 					// Stan bezpiecznego zatrzymania (po Abortingu) 
			
			bServoONRC							:= FALSE;
			bRunProgramRC						:= FALSE;
			bResetErrorRC						:= FALSE;		
			IF bEStop THEN
				eState 				:= E_Station.ePreparingToReady;
				iCaseInit			:=0;
				eRunningState		:=	E_RobotMovState.eReadyPlace;	
			//iActualCase			:= iActualLastCase;
				//IF iActualLastCase = 200 THEN
				//	iActualCase := 250;
				//END_IF
			END_IF
			
	/////////////////////////////	
		E_Station.eAborting:                 	// Stan bezpiecznego zatrzymywania (po EStopie)
			eState 					:=	E_Station.eAborted;  
			iActualLastCase			:=	iActualCase;
		
			
	/////////////////////////////			
		E_Station.eError:                 	 	// Stan błędu 	
	
			iCaseInit				:= 0;
			//bServoONRC			:= FALSE;
			bManualPick			:= FALSE;
			bManualPick2			:= FALSE;
			bManualPlace1				:= FALSE;
			bManualPlace2					:= FALSE;
			
			IF bReset THEN
				eState 				:= E_Station.eResetting;
			END_IF
			
			IF NOT bError THEN
				eState 				:=	E_Station.ePreparingToReady;
				iCaseInit			:=0;
			END_IF
			
	/////////////////////////////
		E_Station.eResetting:					// Stan resetowania bledu (po Errorze)
			
			IF bError THEN
				
				bResetErrorRC					:= bReset;
				eRunningState					:= E_RobotMovState.eReadyPlace;
				bHomingDone						:= FALSE;
				udiErrorId						:= 0;
			END_IF
				
			IF NOT bErrorRCActive  THEN
				bError							:= FALSE;
				bResetErrorRC					:= FALSE;
				bErrorNumberRequest				:= FALSE;				
			END_IF
			
			IF NOT bError THEN
				udiErrorId 			:=	0;
   				sErrorDescription1 	:=	'';
   				sErrorDescription2 	:=	'';				
				eState 				:=	E_Station.ePreparingToReady;
				eRunningState		:=	E_RobotMovState.eReadyPlace;
				iCaseInit			:=0;
//			ELSE
//				eState 				:=	E_Station.eError;
			END_IF
        
	/////////////////////////////
		E_Station.eManualMovement:     			// Stan ruchów manualnych  
       
			ManualMovements();
			//Wyjście z trybu serwisowego
			IF NOT bManualMovement THEN
				eState:=E_Station.eReady;
			END_IF
			IF bHoming THEN
				iCaseHoming					:= 0;
				eState 						:= E_Station.eHoming; 
			END_IF

	/////////////////////////////
		E_Station.eHoming:						// Stan bazowania 
	
			Homing();
			IF NOT bHoming THEN
			   eState:=E_Station.ePreparingToReady;
			   iCaseInit			:=0;
			END_IF		
			
	/////////////////////////////
		E_Station.eHomingDone:                  // Stan wykonania bazowania 
		
			iZ:=iZ+1;
			IF NOT bHoming THEN
			   eState:=E_Station.eReady;
			END_IF
			
	/////////////////////////////
		E_Station.ePreparingToReady:            // Stan przygotowywania do gotowosci (zawsze przed Ready)  
			iCaseRC								:= 0;
			Init();
			
			
	/////////////////////////////
		E_Station.ePreparingToDisable:          // Stan przygotowywania do nieaktywnosci (po wyłączeniu Enable) 
  	
				eState:=E_Station.eDisabled;
			
	/////////////////////////////
		E_Station.eReady:						// Stan gotowosci 
		
			bServoONRC							:= TRUE;
			
			IF bServoONRCActive THEN
				bRunProgramRC					:= TRUE;			
			END_IF
		
			IF bRun AND NOT bCycleDone AND NOT bCycleNotDone THEN
				eState 						:= E_Station.eStarting; 
			END_IF
			
			
			IF bManualMovement AND bRunProgramRC THEN
				//Jeśli przejście w tryb ruchów manualnych przepisz wszystkie stany siłowników sterowanych przez moduł
				//aby zapobiec ewentualnym kolizjom po wejściu w tryb serwisowy
				iCaseManual					:= 0;
				eState 						:= E_Station.eManualMovement; 
			END_IF
			
			IF NOT bRun THEN
				bCycleDone 					:= FALSE;
				bCycleNotDone 				:= FALSE;			
			END_IF
			
			
			IF bHoming THEN
				iCaseHoming					:= 0;
				eState 						:= E_Station.eHoming; 
			END_IF
			
			
			iCaseRC							:= 0;			//22.07.2020
			
			//eRunningState					:=	E_RobotMovState.eReadyPlace;
			
			
		
			
	/////////////////////////////
		E_Station.eStopping:					// Stan zatrzymywania 

			eState 							:= E_Station.eReady;	
			
	/////////////////////////////
		E_Station.eStarting:                  	// Stan uruchamiania (po Ready)	
			bResetErrorRC					:= FALSE;	
			eState					 		:= E_Station.eRunning; 
			
	/////////////////////////////
		E_Station.eRunning:               		// Stan wykonywania cyklu (po Startingu), w tym stanie osobny
 

			IF NOT bRun AND NOT bCycleDone THEN					(*Przerywanie cyklu*)
				eState 				 		:= E_Station.eStopping;	
			END_IF
			
			IF bCycleDone OR bCycleNotDone THEN (*Cykl zakończony*)
				eState 				 		:= E_Station.eReady;
				eRunningState						:=	E_RobotMovState.eReadyPlace;
			END_IF		
			
			Running();
			
			
	/////////////////////////////		
	END_CASE
END_ACTION

ACTION DataExchange:


//SignalOutput
aDataRobotIOOut[1].0                	:= bOperationEnableRC;
aDataRobotIOOut[1].1                	:= bRunProgramRC;
aDataRobotIOOut[1].2              		:= bSlowMotion;
aDataRobotIOOut[1].3                	:= bProgramResetRC;
aDataRobotIOOut[1].4                	:= bServoONRC;
aDataRobotIOOut[1].5                	:= bServoOFFRC;
aDataRobotIOOut[1].6                	:= bResetErrorRC OR bResetWarningRC;
aDataRobotIOOut[1].7                	:= bEditOffset;
aDataRobotIOOut[2].0                	:= bManualCatch;
aDataRobotIOOut[2].1                	:= bErrorNumberRequest OR bWarningNumberRequest;
//Dodane Darek
aDataRobotIOOut[2].7                	:= bBatteryReplacementDone;		//6015
aDataRobotIOOut[3].0                	:= bGreaseReplacementDone;		//6016
aDataRobotIOOut[3].1                	:= bBeltReplacementDone;		//6017
aDataRobotIOOut[3].2                	:= bBeltReplacementDone;		//6017

//SignalRegOutput
aDataRobotREGOut[1]                    	:= INT_TO_UINT(iCaseRC);
aDataRobotREGOut[2]                    	:= INT_TO_UINT(iSpeedSend);
aDataRobotREGOut[3]                    	:= INT_TO_UINT(iPickOffsetX);
aDataRobotREGOut[4]                    	:= INT_TO_UINT(iPickOffsetY);
aDataRobotREGOut[5]                    	:= INT_TO_UINT(iPickOffsetZ);
aDataRobotREGOut[6]                    	:= INT_TO_UINT(iPlace1OffsetX);
aDataRobotREGOut[7]                  	:= INT_TO_UINT(iPlace1OffsetY);
aDataRobotREGOut[8]                    	:= INT_TO_UINT(iPlace1OffsetZ);
aDataRobotREGOut[9]                    	:= INT_TO_UINT(iPlace2OffsetX);
aDataRobotREGOut[10]                	:= INT_TO_UINT(iPlace2OffsetY);
aDataRobotREGOut[11]                	:= INT_TO_UINT(iPlace2OffsetZ);
//Dodane Darek
aDataRobotREGOut[12]                    := INT_TO_UINT(iPick2OffsetX);
aDataRobotREGOut[13]                    := INT_TO_UINT(iPick2OffsetY);
aDataRobotREGOut[14]                    := INT_TO_UINT(iPick2OffsetZ);

// IODATA

fbIntTo2Byte(
iInput:= UDINT_TO_INT(udiIoDATARCWrite), 
byStarszy=> , 
byMlodszy=> );


aDataRobotIOOut[8]												:= fbIntTo2Byte.byStarszy;
aDataRobotIOOut[7]												:= fbIntTo2Byte.byMlodszy;

// Testowy odczyt wartosci wysyłanej
IODATATest                                	:= WORD_TO_UDINT(F_2Bytes_To_Word(aDataRobotIOOut[8], aDataRobotIOOut[7]));


//SignalInput                               
bOperationEnableRCActive            	:= aDataRobotIOIn[1].0;		//6000
bRunProgramRCActive                   	:= aDataRobotIOIn[1].1;
//                                    	:= aDataRobotIOIn[1].2;
bProgramSelectRCActive                	:= aDataRobotIOIn[1].3;
bServoONRCActive                    	:= aDataRobotIOIn[1].4;
bServoOFFRCActive                    	:= aDataRobotIOIn[1].5;
bErrorRCActive                        	:= aDataRobotIOIn[1].6;
bReadyRC                            	:= aDataRobotIOIn[1].7;
bSafePositionRC                        	:= aDataRobotIOIn[2].0;		//6008
bErrorNumberRequestActive               := aDataRobotIOIn[2].1;
bCatcherCloseSensor                    	:= aDataRobotIOIn[2].2;

//Dodane Darek
bHighLevelErrorRCActive                 := aDataRobotIOIn[2].3;		//6011
bLowLevelErrorRCActive                  := aDataRobotIOIn[2].4;		//6012
bWarningRCActive                    	:= aDataRobotIOIn[2].5;		//6013
bBatteryLowVoltage              		:= aDataRobotIOIn[2].6;		//6014
bBatteryReplenishmentFinished               := aDataRobotIOIn[2].7;		//6015
bGreaseReplenishmentFinished	            := aDataRobotIOIn[3].0;		//6016
bBeltReplenishmentFinished	                := aDataRobotIOIn[3].1;		//6017



//SignalRegInput
iActualCase                            	:= UINT_TO_INT(aDataRobotREGIn[1]);
aLoadAxis[0]                        	:= UINT_TO_INT(aDataRobotREGIn[2]);
aLoadAxis[1]                        	:= UINT_TO_INT(aDataRobotREGIn[3]);       
aLoadAxis[2]                        	:= UINT_TO_INT(aDataRobotREGIn[4]);       
aLoadAxis[3]                        	:= UINT_TO_INT(aDataRobotREGIn[5]);
IODATA                                	:= WORD_TO_UDINT(F_2Bytes_To_Word(aDataRobotIOIn[8], aDataRobotIOIn[7]));
END_ACTION

ACTION ErrorDescription:
IF bErrorRCActive AND bHighLevelErrorRCActive THEN

		CASE udiHighLevelErrorId OF	
			
			
0001:					
					
	sErrorDescription1 := 'Fail safe error (SRVOFF).  System problem.';				
	sErrorDescription2 := 'Turn the power OFF and ON once. When it comes back, contact to the dealer.';				
					
0002:					
					
	sErrorDescription1 := 'Fail safe error (STOP).  System Problem.';				
	sErrorDescription2 := 'Turn the power OFF and ON once. When it comes back, contact to the dealer.';				
					
0003:					
					
	sErrorDescription1 := 'System fail.  System Problem.';				
	sErrorDescription2 := 'Check System.When it comes back, contact to the dealer.';				
					
0004:					
					
	sErrorDescription1 := 'CPU Watch dog error.  CPU was not normally treatable.';				
	sErrorDescription2 := 'It is necessary to change some parts when not improvement';				
					
0005:					
					
	sErrorDescription1 := 'Turn the power OFF and ON onc.  The robot model was selected..';				
	sErrorDescription2 := 'Turn the power OFF and ON once';				
					
0006:					
					
	sErrorDescription1 := ' CPU process error.  CPU was not normally treatable.';				
	sErrorDescription2 := 'It is necessary to change some parts when not improvement';				
					
0008:					
					
	sErrorDescription1 := ' CPU synchronization error.  CPU synchronization was failed.';				
	sErrorDescription2 := 'Turn the power OFF and ON once';				
					
0009:					
					
	sErrorDescription1 := 'Version UP (ALL).  Version UP (ALL).';				
	sErrorDescription2 := 'Turn the power OFF,ROTSW=0 and power ON once';				
					
0010:					
					
	sErrorDescription1 := 'Illeagal Version (file).  Version is different.';				
	sErrorDescription2 := 'File was initialized';				
					
0011:					
					
	sErrorDescription1 := 'Illeagal Version (system data.  Version is different.';				
	sErrorDescription2 := 'System data was initialized';				
					
0012:					
					
	sErrorDescription1 := 'Initialize (error log).  Version is different or illegal log file.';				
	sErrorDescription2 := 'Error log was initialized';				
					
0014:					
					
	sErrorDescription1 := 'System error (illegal MECHA).  System error (illegal MECHA).';				
	sErrorDescription2 := 'Set the correct MECHA';				
					
0015:					
					
	sErrorDescription1 := 'Illeagal Version (file).  System ERROR 1.';				
	sErrorDescription2 := 'Contact the maker.';				
					
0016:					
					
	sErrorDescription1 := 'Turn the power OFF and ON onc.  Power OFF/ON a little more slowly,please.';				
	sErrorDescription2 := 'Turn the power OFF and ON once';				
					
0017:					
					
	sErrorDescription1 := '  EEPROM error.  EEPROM is broken.';				
	sErrorDescription2 := 'It is necessary to replace the CPU board';				
					
0019:					
					
	sErrorDescription1 := 'Illegal RotSW on CPU.  RotSW is set not 0.';				
	sErrorDescription2 := 'Please set RotSW to 0';				
					
0020:					
					
	sErrorDescription1 := 'System Error(same name is Bac.  System Error(same name is Backup data.).';				
	sErrorDescription2 := 'Change the system software';				
					
0021:					
					
	sErrorDescription1 := 'System Error(Backup data is C.  System Error(Backup data is Count over.).';				
	sErrorDescription2 := 'Change the system software';				
					
0022:					
					
	sErrorDescription1 := 'System Error(Backup data is n.  System Error(Backup data is no area.).';				
	sErrorDescription2 := 'Change the system software';				
					
0025:					
					
	sErrorDescription1 := ' Files will be saved to ROM.  Program and parameter files will be saved to ROM.';				
	sErrorDescription2 := 'Turn the power OFF and power ON once';				
					
0026:					
					
	sErrorDescription1 := ' Files will be loaded from ROM.  Program and parameter files will be loaded from ROM.';				
	sErrorDescription2 := 'Turn the power OFF and power ON once';				
					
0027:					
					
	sErrorDescription1 := ' Backup or restore is canceled.  Backup or restore is canceled.';				
	sErrorDescription2 := 'Turn the power OFF and power ON once';				
					
0028:					
					
	sErrorDescription1 := ' Memory error (ECC).  2bit error of ECC was detected.';				
	sErrorDescription2 := 'Turn the power OFF and ON once';				
					
0039:					
					
	sErrorDescription1 := 'Door Switch Signal line is fa.  Door Switch Signal line is faulty..';				
	sErrorDescription2 := 'Check the Door Switch Signal line';				
					
0040:					
					
	sErrorDescription1 := 'Door Switch Signal is Input.  Door Switch is opened.';				
	sErrorDescription2 := 'Please close the Door be connected with Door Switch';				
					
0041:					
					
	sErrorDescription1 := 'Comm. error (Remote I/O #1).  Communication line is illegal.';				
	sErrorDescription2 := 'Check the cable or power supply';				
					
0042:					
					
	sErrorDescription1 := ' Comm. error (Remote I/O #2).  Communication line is illegal.';				
	sErrorDescription2 := 'Check the cable or power supply';				
					
0043:					
					
	sErrorDescription1 := ' Comm. error (Remote I/O #3).  Communication line is illegal.';				
	sErrorDescription2 := 'Check the cable or power supply';				
					
0044:					
					
	sErrorDescription1 := ' Comm. error (Remote I/O #4).  Communication line is illegal.';				
	sErrorDescription2 := 'Check the cable or power supply';				
					
0045:					
					
	sErrorDescription1 := ' Comm. error (Remote I/O #5).  Communication line is illegal.';				
	sErrorDescription2 := 'Check the cable or power supply';				
					
0046:					
					
